(* CoDeSys 2.3 export: V4500306_ORIGINAL.EXP *)
(* Libraries: ConnectionDiagnose.lib 3.7.07 16:35:00, PLC_EposCmd.lib 23.7.04 12:26:00, STANDARD.LIB 5.6.98 12:03:02, TcBase.lib 14.5.09 12:14:08, TcBaseMath.lib 27.7.04 12:07:56, TcIoFunctions.lib 27.1.17 17:22:22, TcMath.lib 23.9.04 15:15:30, TcMC.lib 27.7.15 08:51:38, TcNC.lib 10.10.08 17:55:34, TcSystem.lib 7.6.16 11:01:22, TcUtilities.lib 3.2.16 16:08:58 *)

(* Task configuration *)
TASK Standard (PRIORITY := 0, INTERVAL := T#5ms);
PRG_STARTUP();
PRG_VISU();
PRG_PROCESS();
PRG_STATION();
PRG_HW_GENERAL();
PRG_HW_STATION();
PRG_TWINSAFE();
END_TASK
TASK Ctrl_Panel (PRIORITY := 1, INTERVAL := T#100ms);
PRG_USB_IO_PANEL();
END_TASK

(* Global variable list: Constant_Variablen *)
VAR_GLOBAL CONSTANT
	(* developpement *)
	(*sRootPLC:STRING(255):='C:';*)
	(* machine *)
	cssRootPLC:STRING(255):='';
	(* HDD *)
	csiMaxFileLine:INT:=255;
	(* Axis *)
	csiMaxAxisFileObj:INT:=50;
	ciMaxWireStretch:INT:=32767;
	(* Visualisation *)
	csiMaxPage:INT:=50;
	csiMaxUserLevel:INT:=3;
	(* Profile *)
	csiMaxProfile:INT:=100;
END_VAR

(* Global variable list: Globale_Variablen *)
VAR_GLOBAL
(* Structure layer 2 *)
	T_HDD:ST_HDD;
	T_NovRam : ST_NOVRAM;
	T_CtrlePanel:ST_CTRLEPANEL;
	T_DeviceID:ST_DEVICEID;
	T_BoxID:ST_BOXID;
	 T_AxisNodeState AT %I* :ST_NODESTATE;
(* Visualization *)
	QVisCtrl :ST_QVISCTRLE;(*~	(QVis) (InOut:2)	~*)
	T_ExchgParam :ST_QVIS_EXCHG_PARAM;(*~	(QVis) (InOut:2)	~*)
	T_VisuQVis:ST_QVIS;
(* Control Button Start/Stop *)
	T_CtrleBtStartStop:ST_CTRLEBUTTON;
(* StartUp *)
	T_StartUp:ST_STARTUP;
(* Station *)
	T_Station:ST_STATION;
(* Process *)
	T_Process : ST_PROCESS;
(* Profile *)
	T_Profile:ST_PROFILE;
(* Static Error List *)
	T_ErrorList:ST_ERROR_LIST;	(* Static define Error List *)
(* IO's *)
	IarxDigitalInput AT %I* : ARRAY[1..64] OF BOOL;
	QarxDigitalOutput AT %Q* : ARRAY[1..64] OF BOOL;
	IariAnalogInput AT %I* : ARRAY[1..32] OF INT;
	QariAnalogOutput AT %Q* : ARRAY[1..32] OF INT;
	QarxCylinder AT %Q* : ARRAY[1..32] OF BOOL;
(* TwinSafe *)
	T_TwinSafeCtrleIN AT %I*:ST_TWINSAFE_CTRLE_IN;
	T_TwinSafeCtrleOUT AT %Q*:ST_TWINSAFE_CTRLE_OUT;
	T_TwinSafeIn:ST_TWINSAFE_IN;
	T_TwinSafeOut AT %I*:ST_TWINSAFE_OUT;
END_VAR

(* Global variable list: TwinCAT_Configuration *)
(* Generated automatically by TwinCAT - (read only) *)
VAR_CONFIG
	PRG_HW_STATION.TToolLeftRxPdoPara AT %QB0 : ST_RX_PDO_PARA;
	PRG_HW_STATION.TToolLeftTxPdoPara AT %IB0 : ST_TX_PDO_PARA;
	PRG_HW_STATION.TToolCenterRxPdoPara AT %QB27 : ST_RX_PDO_PARA;
	PRG_HW_STATION.TToolCenterTxPdoPara AT %IB17 : ST_TX_PDO_PARA;
	PRG_HW_STATION.TToolRightRxPdoPara AT %QB54 : ST_RX_PDO_PARA;
	PRG_HW_STATION.TToolRightTxPdoPara AT %IB34 : ST_TX_PDO_PARA;
	PRG_HW_STATION.TToolFeederRxPdoPara AT %QB81 : ST_RX_PDO_PARA;
	PRG_HW_STATION.TToolFeederTxPdoPara AT %IB51 : ST_TX_PDO_PARA;
	PRG_HW_STATION.TGrindFeederRxPdoPara AT %QB108 : ST_RX_PDO_PARA;
	PRG_HW_STATION.TGrindFeederTxPdoPara AT %IB68 : ST_TX_PDO_PARA;
	PRG_HW_STATION.stToolLeftRefOut AT %QB135 : PLCTONC_AXLESTRUCT;
	PRG_HW_STATION.stToolLeftRefIn AT %IB85 : NCTOPLC_AXLESTRUCT;
	PRG_HW_STATION.stToolCenterRefOut AT %QB263 : PLCTONC_AXLESTRUCT;
	PRG_HW_STATION.stToolCenterRefIn AT %IB213 : NCTOPLC_AXLESTRUCT;
	PRG_HW_STATION.stToolRightRefOut AT %QB391 : PLCTONC_AXLESTRUCT;
	PRG_HW_STATION.stToolRightRefIn AT %IB341 : NCTOPLC_AXLESTRUCT;
	PRG_HW_STATION.stToolFeederRefOut AT %QB519 : PLCTONC_AXLESTRUCT;
	PRG_HW_STATION.stToolFeederRefIn AT %IB469 : NCTOPLC_AXLESTRUCT;
	PRG_HW_STATION.stGrindFeederRefOut AT %QB647 : PLCTONC_AXLESTRUCT;
	PRG_HW_STATION.stGrindFeederRefIn AT %IB597 : NCTOPLC_AXLESTRUCT;
	PRG_HW_STATION.auiActualAxisTorqueBeckhoff AT %IB725 : ARRAY [1..5] OF UINT;
	PRG_HW_STATION.axInputAxisBeckhoff AT %IB735 : ARRAY [1..5, 1..8] OF BOOL;
	PRG_TWINSAFE.TwinSAFEinputKlemme1.KLx904_SafetyIn AT %IB920 : TwinSAFE_SafetyIn;	(*  ~ {LinkedWith:TIID^CX1000_PLC^CX1100-KB^Klemme 9 (KL1904)^Kanal 1^Safety In} *)
	PRG_TWINSAFE.TwinSAFEinputKlemme2.KLx904_SafetyIn AT %IB926 : TwinSAFE_SafetyIn;	(*  ~ {LinkedWith:TIID^CX1000_PLC^CX1100-KB^Klemme 10 (KL1904)^Kanal 1^Safety In} *)
	PRG_TWINSAFE.TwinSAFEinputKlemme3.KLx904_SafetyIn AT %IB932 : TwinSAFE_SafetyIn;	(*  ~ {LinkedWith:TIID^CX1000_PLC^CX1100-KB^Klemme 11 (KL1904)^Kanal 1^Safety In} *)
	PRG_USB_IO_PANEL.IarxCtrlePanelButton AT %IB775 : ARRAY [1..10] OF BOOL;
	PRG_USB_IO_PANEL.QarxCtrlePanelLed AT %QB775 : ARRAY [1..10] OF BOOL;
	.T_AxisNodeState AT %IB940 : ST_NODESTATE;
	.IarxDigitalInput AT %IB785 : ARRAY [1..64] OF BOOL;
	.QarxDigitalOutput AT %QB785 : ARRAY [1..64] OF BOOL;
	.IariAnalogInput AT %IB849 : ARRAY [1..32] OF INT;
	.QariAnalogOutput AT %QB849 : ARRAY [1..32] OF INT;
	.QarxCylinder AT %QB913 : ARRAY [1..32] OF BOOL;
	.T_TwinSafeCtrleIN AT %IB913 : ST_TWINSAFE_CTRLE_IN;
	.T_TwinSafeCtrleOUT AT %QB945 : ST_TWINSAFE_CTRLE_OUT;
	.T_TwinSafeOut AT %IB916 : ST_TWINSAFE_OUT;
END_VAR

(* Data type in AXIS *)
TYPE ST_AXIS :
STRUCT
	T_CtrleSingle:ST_CTRLESINGLE;
	T_CtrleMulti:ST_CTRLEMULTI;
	T_ParamFileObj:ARRAY[1..40] OF ST_PARAM_FILE_OBJ;
	T_Config_Gen:ST_CONFIG_GENERAL;
	T_Config_ObjFileValue:ST_CONFIG_OBJECT;	(* Gilt nicht für Ecostep *)
 	T_Config_Setting:ST_CONFIG_SETTING;			(* Gilt nicht für Ecostep *)
	T_LiveValue:ST_LIVEVALUE;
	T_Oscillation:ST_OSCILLATION;					(* Gilt nicht für Ecostep *)
	T_Torque:ST_AXISTORQUE;					(* Gilt nicht für Ecostep *)
	T_FileObj:ST_AXIS_FILE_OBJ;
	T_RxPdoParameter:ST_RX_PDO_PARA;
	T_TxPdoParameter:ST_TX_PDO_PARA;
	T_SoftwareDetails:ST_SOFTWARE_INFO;
END_STRUCT
END_TYPE

(* Data type in AXIS *)
TYPE ST_AXIS_FILE_OBJ :
STRUCT
	sData: ARRAY[1..csiMaxAxisFileObj] OF STRING(120);
END_STRUCT
END_TYPE

(* Data type in AXIS *)
TYPE ST_AXISTORQUE :
STRUCT
(* input *)
	xActive:BOOL;
(* output *)
	rAverage:REAL;
	rMinAverage:REAL;
	rMaxAverage:REAL;
	rLastValue:REAL;
	rMinValue:REAL;
	rMaxValue:REAL;
	iSensitivity:INT;
	rMaxVariationSpindle:REAL;
	rActualVariationSpindle:REAL;
END_STRUCT
END_TYPE

(* Data type in AXIS *)
TYPE ST_CONFIG_GENERAL :
STRUCT
	sDeviceName:STRING(32);
	sDeviceFileName:STRING(32);
	sFileNamePDOMapping:STRING(32);
	sServoNetId:STRING(23);		(* Beckhoff *)
	sAmsNetId:T_AmsNetId;		(* Ecostep *)
	udiNC_TaskIdxGrp:UDINT;		(* Beckhoff *)
	udiNodeId:UDINT;				(* Ecostep *)
	iTyp:INT;
	iMachineType:INT;			(* 1 = MicroWire, 2 = MicroRod *)
END_STRUCT
END_TYPE

(* Data type in AXIS *)
TYPE ST_CONFIG_OBJECT :
STRUCT
(* Object value *)
	lrMaxVelocity:LREAL;
	lrCalVelocityForward:LREAL;
	lrCalVelocityBackward:LREAL;
	lrAcceleration:LREAL;
	lrDecceleration:LREAL;
	lrJerk:LREAL;
	xSWLimitPos:BOOL;
	xHWLimitPos:BOOL;
	lrSWLimitPos:LREAL;
	xSWLimitNeg:BOOL;
	xHWLimitNeg:BOOL;
	lrSWLimitNeg:LREAL;
	lrScaleFactor:LREAL;
END_STRUCT
END_TYPE

(* Data type in AXIS *)
TYPE ST_CONFIG_SETTING :
STRUCT
	lrJogFast:LREAL;
	lrJogSlow:LREAL;
	lrJogStepFast:LREAL;
	lrJogStepSlow:LREAL;
	lrVelocityAbs:LREAL;
	lrVelocityRel:LREAL;
	lrVelocityProcess:LREAL;
	lrSpindleCurrentLimit:LREAL;
	xHardwareLimitPos:BOOL;
	xHardwareLimitNeg:BOOL;
	lrHWLimitDecceleration:LREAL;
	rHCRampDeceleration:REAL;
	rHCRampJerk:REAL;
END_STRUCT
END_TYPE

(* Data type in AXIS *)
TYPE ST_CTRLEMULTI :
STRUCT
(* Input *)
	xExecute:BOOL:=FALSE;
	xReset:BOOL:=FALSE;
	iNumerator:INT:=1;
	uiDenominator:UINT:=1;
	iFunction:INT:=0;

(* Ouput *)
	xDone:BOOL:=FALSE;
	xErr:BOOL:=FALSE;
	udiErrorID:UDINT:=0;
END_STRUCT
END_TYPE

(* Data type in AXIS *)
TYPE ST_CTRLESINGLE :
STRUCT
(* Input *)
	xExecute:BOOL:=FALSE;
	iFunction:INT:=0;
	xReset:BOOL:=FALSE;
	iInput:INT:=0;
	lrPosition:LREAL:=0;
	lrDistance:LREAL:=0;
	lrVelocity:LREAL:=0;
	lrAcceleration:LREAL:=0;
	lrDecceleration:LREAL:=0;
	lrJerk:REAL:=0;
	dwOverride:DWORD:=100;
	rSetPosition:REAL:=0;
	rSetTorque:REAL:=0;
	sSend:STRING(20):='';
	lrScaleFactor:LREAL:=0;
	lrGearRatioFactor:LREAL:=0;
	lrGearRatioDivider:LREAL:=0;
	lrGearRatio:LREAL:=0;	(* calculate lrGearRatioFactor / lrGearRatioDivider *)
	iModuloDirection:INT;		(*	Enum Werte:
									 MC_Positive_Direction := 1,
    									MC_Shortest_Way :=2,
    									MC_Negative_Direction :=3,
    									MC_Current_Direction :=4
							*)
	lrHomingMethode:LREAL;
	lrHomeOffset:LREAL;
	lrHomeSpeedSwitch:LREAL;
	lrHomeSpeedZero:LREAL;
	lrHomeAcceleration:LREAL;
	lrGearFactor:LREAL;
	lrGearDivider:LREAL;
	lrSWNegLimitSwitch:LREAL;
	lrSWPosLimitSwitch:LREAL;
	xBlockAcclDeclParameter:BOOL;

(* Output *)
	xDone:BOOL:=FALSE;
	xErr:BOOL:=FALSE;
	udiErrorID:UDINT:=0;
	xPower:BOOL:=FALSE;
	xReady:BOOL:=FALSE;
	xNotMoving:BOOL:=FALSE;
	xRef:BOOL:=FALSE;
	xSlave:BOOL:=FALSE;
	xConstantVel:BOOL:=FALSE;
	xBusyNewPosAndVel:BOOL:=FALSE;
	xDriveTorque:BOOL:=FALSE;
	iOutput:INT:=0;
	xSWLimitPos:BOOL:=FALSE;
	xSWLimitNeg:BOOL:=FALSE;
	xHWLimitPos:BOOL:=FALSE;
	xHWLimitNeg:BOOL:=FALSE;
	xSpindleBlocked:BOOL:=FALSE;
	iStrokeAngleRefIndex:INT;	(* Gilt für die Prozedur für das einstellen des Referenzindex der Achse *)
END_STRUCT
END_TYPE

(* Data type in AXIS *)
TYPE ST_LIVEVALUE :
STRUCT
	dwState:DWORD;
	uiActualTorque:UINT;
	diActualTorqueCalc:DINT;	(* entsricht dem uiActualTorque, nur dass positiver und negativer Torque berücksichtigt wird *)
	lrActualVelocity:LREAL;
	lrActualPosition:LREAL;
	bDigitalInput:BYTE;
	lrSollPosition:LREAL;
	lrActualPositionNotModulo:LREAL;
	lrActualPositionRelativ:LREAL;
END_STRUCT
END_TYPE

(* Data type in AXIS *)
TYPE ST_NODESTATE :
STRUCT
	bToolLeftNodeState:BYTE;
	bToolCenterNodeState:BYTE;
	bToolRightNodeState:BYTE;
	bToolFeederNodeState:BYTE;
	bGrindFeederNodeState:BYTE;
END_STRUCT
END_TYPE

(* Data type in AXIS *)
TYPE ST_OSCILLATION :
STRUCT
	rFrequence:REAL;
	rOffset:REAL;
	rPosTorqueLimitOffset:REAL;
	iCycle:INT;
END_STRUCT
END_TYPE

(* Data type in AXIS *)
TYPE ST_PARAM_FILE_OBJ :
STRUCT
	udiIdxGroup:UDINT:=0;
	udiIndexOffset:UDINT:=0;
	udiLength:UDINT:=0;
	lrReal:LREAL:=0;
	sName:STRING(20);
END_STRUCT
END_TYPE

(* Data type in AXIS *)
TYPE ST_RX_PDO_PARA :
STRUCT
	udiProfileVelocity:UDINT;
	diTargetVelocity:DINT;
	udiProfileDeceleration:UDINT;
	udiProfileAcceleration:UDINT;
	diTargetPosition:DINT;
	iGearFactor:INT;
	uiGearDivider:UINT;
	iControlWord:INT;
	siOperationModes:SINT;
END_STRUCT
END_TYPE

(* Data type in AXIS *)
TYPE ST_SOFTWARE_INFO :
STRUCT
	lrSoftwareVersion:REAL;
	lrBuildVersion:REAL;
	lrDateCode:REAL;
	sDateCode:STRING;
END_STRUCT
END_TYPE

(* Data type in AXIS *)
TYPE ST_TX_PDO_PARA :
STRUCT
	diActualPosition:DINT;
	diActualVelocity:DINT;
	uiStatusWord:UINT;
	iActualCurrent:INT;
	udiDigitalInput:UDINT;
	siOperationModesDisplay:SINT;
END_STRUCT
END_TYPE

(* Data type in CX1020 *)
TYPE ST_BOXID :
STRUCT
(* control structure *)
	T_Ctrle:ST_CTRLE_DEVICEID;
(* Data *)
	(* servo Beckhoff-->Lightbus *)
	T_Servo_ToolLeft:ST_BOXID_DATA_ADR;
	T_Servo_ToolCenter:ST_BOXID_DATA_ADR;
	T_Servo_ToolRight:ST_BOXID_DATA_ADR;
	T_Servo_ToolFeeder:ST_BOXID_DATA_ADR;
	T_Servo_GrindFeeder:ST_BOXID_DATA_ADR;
END_STRUCT
END_TYPE

(* Data type in CX1020 *)
TYPE ST_BOXID_DATA_ADR :
STRUCT
	sDeviceName:T_MaxString;
	sBoxName:T_MaxString;
	xDeviceOption:BOOL;
	wAddrBox:WORD;
	sAmsNetId:T_AmsNetId;
END_STRUCT
END_TYPE

(* Data type in CX1020 *)
TYPE ST_CTRLE_DEVICEID :
STRUCT
(* input *)
	xExecute:BOOL:=FALSE;
	xReset:BOOL:=FALSE;
	xLocked:BOOL:=FALSE;
(*
	iStationNr:INT:=0;
	iStationType:INT:=0;
	iSpindleType:INT:=0;
*)
	iMachineType:INT:=0;

(* output *)
	xDone:BOOL:=FALSE;
	xErr:BOOL:=FALSE;
	udiErrorID:UDINT:=0;

END_STRUCT
END_TYPE

(* Data type in CX1020 *)
TYPE ST_DEVICEID :
STRUCT
(* control structure *)
	T_Ctrle:ST_CTRLE_DEVICEID;
(* Data *)
	(* PLC *)
		T_CX1020:ST_DEVICEID_DATA_ADR;
	(* feldbus *)
		T_CANOpenMaster:ST_DEVICEID_DATA_ADR;
		T_LightbusMaster:ST_DEVICEID_DATA_ADR;
	(* NovRAM *)
		T_NovRAM:ST_DEVICEID_DATA_ADR;
END_STRUCT
END_TYPE

(* Data type in CX1020 *)
TYPE ST_DEVICEID_DATA_ADR :
STRUCT
	sDeviceName:T_MaxString;
	xDeviceOption:BOOL;
	udiDeviceID:UDINT;
	sAmsNetId:T_AmsNetId;
END_STRUCT
END_TYPE

(* Data type in Cylinder *)
TYPE ST_ANALOG :
STRUCT
(* input *)
	tDelayActiv:TIME;
	iAnalogIN:INT;
	rForceIn:REAL;
	iRampFctOn:INT;
	iRampFctOff:INT;
	rStepValue:REAL;
	rLengthIn:REAL;
(* Output *)
	xActiv:BOOL;
	iAnalogOut:INT;
	rForceOut:REAL;
	tTimeActivOn:TIME;
	tTimeActivOff:TIME;
END_STRUCT
END_TYPE

(* Data type in Cylinder *)
TYPE ST_ANALOG_CYL :
STRUCT
(* input *)
	tDelayActiv:TIME;
	iAnalogIN:INT;
	rForceIn:REAL;
(* Output *)
	xActiv:BOOL;
	iAnalogOut:INT;
	rForceOut:REAL;
END_STRUCT
END_TYPE

(* Data type in Cylinder *)
TYPE ST_CONFIG :
STRUCT
	tDelayOn:TIME;
	tDelayOff:TIME;
	tDelayPreOn:TIME;
	tDelayPreOff:TIME;
	xCtrlePosOn:BOOL;
	xCtrlePosOff:BOOL;
	tTimeOut:TIME;
	xActivState:BOOL;
END_STRUCT
END_TYPE

(* Data type in Cylinder *)
TYPE ST_CTRLECYL :
STRUCT
(* input *)
	xFBActiv:BOOL;
	xExecute:BOOL;
	xReset:BOOL;
	iFunction:INT;
(* output *)
	xDone:BOOL;
	xErr:BOOL;
	udiErrorID:UDINT;
	xStatePosOn:BOOL;
	xStatePosOff:BOOL;
	T_AnalogCylinder:ST_ANALOG_CYL;
	T_Standard:ST_STANDARD;
	T_Analog:ST_ANALOG;
END_STRUCT
END_TYPE

(* Data type in Cylinder *)
TYPE ST_CYLINDER :
STRUCT
	T_Config:ST_CONFIG;
	T_CtrleCyl:ST_CTRLECYL;
END_STRUCT
END_TYPE

(* Data type in Cylinder *)
TYPE ST_STANDARD :
STRUCT
(* Input *)
	tDelayActiv:TIME;
	tDelayAfterSensor:TIME;
(* Output *)
	xActivOn:BOOL;
	xActivOff:BOOL;
END_STRUCT
END_TYPE

(* Data type in Geometry *)
TYPE ST_GEOMETRY :
STRUCT
	arStartDiameter: ARRAY [1..6] OF REAL;
	arEndDiameter: ARRAY [1..6] OF REAL;
	arSectionLength: ARRAY [1..6] OF REAL;
	arSectionPitch: ARRAY [1..6] OF REAL;
	axActiveSection:ARRAY [1..6] OF BOOL;
END_STRUCT
END_TYPE

(* Data type in Geometry *)
TYPE ST_GEOMETRY_COMMON :
STRUCT
	abSectionSelectForm:ARRAY [1..6] OF BYTE; (* 0=Disactivate Section, 1=Zylindre large, 2=Zylindre small, 3=Cone Negative, 4=Cone Positive *)
	wWrongInput:WORD;
	wWrongInput_2:WORD;
	rMinToolDiameter:REAL;
	rMaxToolDiameter:REAL;
	rMinToolLength:REAL;
	rMaxToolLength:REAL;
	T_Geometry:ST_GEOMETRY;
END_STRUCT
END_TYPE

(* Data type in HDD *)
TYPE ST_CTRLE_HDD :
STRUCT
(* input *)
	xExecute:BOOL:=FALSE;
	xReset:BOOL:=FALSE;
	iFunction:INT:=0;
	tTimeOut:TIME;
	xLocked:BOOL:=FALSE;

(* output *)
	xDone:BOOL:=FALSE;
	xErr:BOOL:=FALSE;
	udiErrorID:UDINT:=0;
END_STRUCT
END_TYPE

(* Data type in HDD *)
TYPE ST_HDD :
STRUCT
	T_Ctrle:ST_CTRLE_HDD;
	T_Config:ST_HDD_CONFIG;
	T_File:ST_HDD_FILE;
	T_Data:ST_HDD_DATA;
END_STRUCT
END_TYPE

(* Data type in HDD *)
TYPE ST_HDD_CONFIG :
STRUCT
	sNetId:T_AmsNetId;
END_STRUCT
END_TYPE

(* Data type in HDD *)
TYPE ST_HDD_DATA :
STRUCT
	sData: ARRAY[1..csiMaxFileLine] OF STRING(255);
END_STRUCT
END_TYPE

(* Data type in HDD *)
TYPE ST_HDD_FILE :
STRUCT
	sPathAndFileName:STRING(255):='';
	sOldPathAndFileName:STRING(255):='';
	dwPtrWriteBuffer:DWORD:=0;
	udiLenBuffer:UDINT:=0;
END_STRUCT
END_TYPE

(* Data type in Panel *)
TYPE ST_CTRLEPANEL :
STRUCT
(* Input *)
	xExecute:BOOL:=FALSE;
	iFunction:INT:=0;
	xReset:BOOL:=FALSE;
(* output *)
	xDone:BOOL;
	xErr:BOOL;
	udiErrorID:UDINT;
	udiButton:UDINT:=0;
	udiLED:UDINT:=0;
END_STRUCT
END_TYPE

(* Data type in Process *)
TYPE ST_FCTPROCESS :
STRUCT
	xEnable : BOOL :=FALSE;
	xStart: BOOL := FALSE;
	xStop: BOOL := FALSE;
	xStopCycle : BOOL :=FALSE;
	xQuitErr : BOOL := FALSE;
	xAbord : BOOL := FALSE;
	xProcessHold : BOOL;
	xEnd : BOOL := FALSE;
	xError : BOOL := FALSE;
	diErrorNr : DINT := 0;
END_STRUCT
END_TYPE

(* Data type in Process *)
TYPE ST_PARA_WARMUP :
STRUCT
	iWarmUp_TimeON_Hour		:INT;
	iWarmUp_TimeON_Minute		:INT;
	iWarmUp_TimeOFF_Hour		:INT;
	iWarmUp_TimeOFF_Minute		:INT;
	axDayOfWeek				:ARRAY [0..7] OF BOOL;	(* 0=Sonntag, 1=Montag..usw *)

(*SOA 30.01.23 *)
	iWarmUp_TimeDIF_Hour		:INT;
	iWarmUp_TimeDIF_Minute		:INT;
END_STRUCT
END_TYPE

(* Data type in Process *)
TYPE ST_PROCESS :
STRUCT
	iFunctNr : INT :=0;
	xEnable : BOOL := FALSE;
	xStart : BOOL := FALSE;
	xEnd : BOOL := FALSE;
	xStop : BOOL := FALSE;
	xStopCycle : BOOL :=FALSE;
	xRdy : BOOL := FALSE;
	xError : BOOL := FALSE;
	diErrorNr : DINT :=0;
	xQuitError : BOOL := FALSE;
	xProcessHold : BOOL;
	wStatus : WORD := 0;
	xAbord : BOOL := FALSE;
	xReferenced : BOOL := FALSE;
	TFctProcess : ST_FCTPROCESS;
END_STRUCT
END_TYPE

(* Data type in Profile *)
TYPE ST_PROFILE :
STRUCT
	T_Ctrle:ST_PROFILE_CTRLE;
	T_Id:ST_PROFILE_ID;
	(*T_DataOnline:ST_PROFILEONLINECHANGE;*)
END_STRUCT
END_TYPE

(* Data type in Profile *)
TYPE ST_PROFILE_CTRLE :
STRUCT
(* input *)
	xExecute:BOOL:=FALSE;
	xReset:BOOL:=FALSE;
	iFunction:INT:=0;

(* Output *)
	xDone:BOOL:=FALSE;
	xErr:BOOL:=FALSE;
	udiErrorID:UDINT:=0;
END_STRUCT
END_TYPE

(* Data type in Profile *)
TYPE ST_PROFILE_ID :
STRUCT
	iNumber:INT;
	sName:STRING(30);
END_STRUCT
END_TYPE

(* Data type in Profile *)
TYPE ST_PROFILE_LIST :
STRUCT
	iNumber:INT;
	sName:STRING(30);
END_STRUCT
END_TYPE

(* Data type in Profile *)
TYPE ST_PROFILE_LIST_MANAGE :
STRUCT
	xListProfileUp:BOOL;
	xListProfileDown:BOOL;
	xListProfileUpFast:BOOL;
	xListProfileDownFast:BOOL;
END_STRUCT
END_TYPE

(* Data type in QVis *)
TYPE ST_BUTTON :
STRUCT
	xInputState:BOOL;
	xLedState:BOOL;
	xResetTime:BOOL;
	tPressTime:TIME;
END_STRUCT
END_TYPE

(* Data type in QVis *)
TYPE ST_CONFIGPAGE :
STRUCT
	sName:STRING(32);
	wMaskBtPanelLeft:WORD;
	wMaskBtPanelRight:WORD;
	wMaskFunctionPanel:WORD;
	wMaskTouchScreenNavPanel:WORD;
	(* active movement mask *)
	wMaskActiveMachineBtPanelLeft:WORD;
	wMaskActiveMachineBtPanelRight:WORD;
	wMaskActiveMachineFunctionPanel:WORD;
	wMaskActiveMachineNavPanel:WORD;
	(* functions *)
	aiRTrigActionPanelRight:ARRAY[1..5] OF INT:=5(0);
	aiFTrigActionPanelRight:ARRAY[1..5] OF INT:=5(0);
	aiDelayActionPanelRight:ARRAY[1..5] OF INT:=5(0);
	aiRTrigActionFunctionPanel:ARRAY[1..12] OF INT:=12(0);
	aiFTrigActionTouchScreenNavPanel:ARRAY[1..6] OF INT:=6(0);
	(* start/stop button *)
	xMaskBtStart:BOOL;
	xMaskBtStop:BOOL;
END_STRUCT
END_TYPE

(* Data type in QVis *)
TYPE ST_CTRLEACTION :
STRUCT
(* Input *)
	xExecute:BOOL;
	xReset:BOOL;
	iFunction:INT;
	xResetParaListValue:BOOL;
(* Output *)
	xDone:BOOL;
	xNotReady:BOOL;
	xErr:BOOL;
	udiErrorID:UDINT;
END_STRUCT
END_TYPE

(* Data type in QVis *)
TYPE ST_CTRLEBUTTON :
STRUCT
	T_Start:ST_BUTTON;
	T_Stop:ST_BUTTON;
END_STRUCT
END_TYPE

(* Data type in QVis *)
TYPE ST_CTRLEPROCESS :
STRUCT
(* Input *)
	xExecute:BOOL;
	xReset:BOOL;
	iFunction:INT;
(* Output *)
	xDone:BOOL;
	xErr:BOOL;
	udiErrorID:UDINT;
END_STRUCT
END_TYPE

(* Data type in QVis *)
TYPE ST_CTRLEVISU :
STRUCT
(* Input *)
	xActive:BOOL;
	xExecute:BOOL;
	xReset:BOOL;
	iFunction:INT;
(* Output *)
	xDone:BOOL;
	xErr:BOOL;
	udiErrorID:UDINT;
	xQvis:BOOL;
END_STRUCT
END_TYPE

(* Data type in QVis *)
TYPE ST_EXCHG_BTFUNCTIONPANEL :
STRUCT
	wState:WORD;
	wActivBt:WORD;
	wNotMasktext:WORD;
	bF1SelectText:BYTE;
	bF2SelectText:BYTE;
	bF3SelectText:BYTE;
	bF4SelectText:BYTE;
	bF5SelectText:BYTE;
	bF6SelectText:BYTE;
	bF7SelectText:BYTE;
	bF8SelectText:BYTE;
	bF9SelectText:BYTE;
	bF10SelectText:BYTE;
	bF11SelectText:BYTE;
	bF12SelectText:BYTE;
END_STRUCT
END_TYPE

(* Data type in QVis *)
TYPE ST_EXCHG_CONFIG :
STRUCT
	xNoTouchScreenBtPanel:BOOL;
	iEditParam:INT;
	xBlockParaListNavi:BOOL;
	xBlockParaListNavi1:BOOL;
	xBlockNavParaList:BOOL;
	xBlockNavParaListTeachRot:BOOL;
	xBlockProfilList:BOOL;
	iSelectParaList:INT;
	iSelectParaListTeachRot:INT;
END_STRUCT
END_TYPE

(* Data type in QVis *)
TYPE ST_EXCHG_CYLINDER :
STRUCT
(*	iSelectCylToolTension:INT; *)
	xToolTension:BOOL;
	bPosToolTension:BYTE;

	T_ParamToolTension:ST_EXCHG_PARAM_CYL_FORCE;
	iSelectToolTensionForce:INT;
	rToSetToolTensionForce:REAL;
(*22.12.2009: KFS	{	*)
	iSelectCylinder_Sonder1:INT;

	xCylToolLeft:BOOL;
	bPosCylToolLeft:BYTE;

	xCylToolRight:BOOL;
	bPosCylToolRight:BYTE;

	xCylToolCenter:BOOL;
	bPosCylToolCenter:BYTE;

	xCylToolPrismaLeft:BOOL;
	bPosCylToolPrismaLeft:BYTE;

	xCylToolPrismaRight:BOOL;
	bPosCylToolPrismalRight:BYTE;
(*22.12.2009: KFS	}	*)
END_STRUCT
END_TYPE

(* Data type in QVis *)
TYPE ST_EXCHG_FUNCTION_COMMON :
STRUCT
	(* Overlay for input measured Tool diameter *)
	xOpenOverlayMeasureInput:BOOL;
	(* Overlay for input the correction of the GrindFeeder Plunge *)
	xOpenOverlaySetGrindPlunge:BOOL;
	(* Overlay for open a Messagebox *)
	xOpenOverlayMessageBox:BOOL;
	sMessageBoxLine1:STRING(50);
	sMessageBoxLine2:STRING(50);
	sMessageBoxLine3:STRING(50);
	sMessageBoxLine4:STRING(50);
	sMessageBoxLine5:STRING(50);
	sMessageBoxLine6:STRING(50);
	xSaveButton:BOOL;
	xExitButton:BOOL;
	rInputMeasToolDiameter:REAL;
	rInputGrindPlunge:REAL;
	xHideProgressbar:BOOL;

	(*SOA 12.01.2023 { *)
	(* Setup WarmUp *)
	TWarmUp_Para						:ST_PARA_WARMUP;
	axWarmUp_DayOfWeekButton			:ARRAY [0..6] OF BOOL;	(* 0=Sonntag, 1=Montag..usw *)
	xWarmUp_ContactorMachine_Active		:BOOL;
	xWarmUp_MessageWarning			:BOOL;	(* Mittels dieser Meldung wird hingewiesen dass die Maschine nächstens eingeschaltet wird *)
	xWarmUp_MessageWarning_2			:BOOL;	(* Mittels dieser Meldung wird gefragt, ob die Maschine wirklich eingeschaltet werden soll *)
	iWarmUp_ColourChange				:BOOL;
	(*SOA 12.01.2023 } *)

END_STRUCT
END_TYPE

(* Data type in QVis *)
TYPE ST_EXCHG_INFO_PROCESS :
STRUCT
	iProfile:INT;
	sProfileName:STRING(30);
	xOnlineValueModified:BOOL;
END_STRUCT
END_TYPE

(* Data type in QVis *)
TYPE ST_EXCHG_INFOVALUE_COMMON :
STRUCT
	rActualGrindAxisPosition:REAL;
	rActualGrindAxisSpeed:REAL;
	rActualToolRotSpeed:REAL;
	rActualWireFeedPosition:REAL;
	rActualWireFeedSpeed:REAL;
	rActualToolLeftTorque:REAL;
	rCalculToolLeftTorque:REAL;
	rActualToolCenterTorque:REAL;
	rCalculToolCenterTorque:REAL;
	rActualToolRightTorque:REAL;
	rCalculToolRightTorque:REAL;
	rToolLengthCalibration:REAL;
	rToolDiameter:REAL;
	rToolTotalLength:REAL;
	rPitchCalibration:REAL;
	rToolTensionForce:REAL;
	iTotalCountDownCycle:INT;
	iCountDownCycle:INT;
	iTotalCountDownPlungeCycle:INT;
	iCountDownPlungeCycle:INT;
	iTotalCountDownGrooveCycle:INT;
	iCountDownGrooveCycle:INT;
	tAutoTimeTotal:TIME;
	tAutoTimeLeft:TIME;

	rCorrectionToolDiameter:REAL;
	xKeyPadActivation:BOOL;

	(* Progressbar for Tool Calibration *)
	bProgressbarToolCalibration:BYTE;
	bProgressbarAutoGeometry:BYTE;
	bProgressbarAutoGroove:BYTE;

	(* Effectiv working geometry *)
	arStartDiameter: ARRAY [1..6] OF REAL;
	arEndDiameter: ARRAY [1..6] OF REAL;
	(* Part State display *)
	bActivePartNumber:BYTE;

END_STRUCT
END_TYPE

(* Data type in QVis *)
TYPE ST_EXCHG_LEVEL :
STRUCT
	iActLevel:INT;
	iPwSystem:INT;
	iRandom:INT;
END_STRUCT
END_TYPE

(* Data type in QVis *)
TYPE ST_EXCHG_MACHINE :
STRUCT
	iFunction:INT;
	udiState_Input:UDINT;
	T_Process:ST_EXCHG_PROCESS;
END_STRUCT
END_TYPE

(* Data type in QVis *)
TYPE ST_EXCHG_MESSAGE :
STRUCT
	iState:INT;
	iStateBIOS:INT;
	sDynamicTextEnglish:STRING(100);
	sDynamicTextDeutsch:STRING(100);
	sDynamicTextFrancais:STRING(100);
END_STRUCT
END_TYPE

(* Data type in QVis *)
TYPE ST_EXCHG_MESSAGE_ERROR :
STRUCT
	asMsgErrorList:ARRAY [1..20] OF STRING(100);
END_STRUCT
END_TYPE

(* Data type in QVis *)
TYPE ST_EXCHG_PARAM_AUTOGEOMETRY :
STRUCT
	rPlungeLengthToolFeedGeometry:REAL;
	rPlungeSpeedGrindFeedGeometry:REAL;
	rDisplaceLengthToolFeedGeometry:REAL;
	rDisplaceSpeedGrindFeedGeometry:REAL;
	xPlungeActivationGeometry:BOOL;
	xDisplaceActivationGeometry:BOOL;
	iCycleGeometry:INT;
	rPlungeCycleGrindFeedGeometry:REAL;
	rSpeedToolRotationGeometry:REAL;
(*08.07.2014: KFS	{	*)
	xWarmUp:BOOL;
(*08.07.2014: KFS	}	*)
	 xMoveTableStuderBW:BOOL;  (*SOA *)
END_STRUCT
END_TYPE

(* Data type in QVis *)
TYPE ST_EXCHG_PARAM_AUTOGROOVE :
STRUCT
	rPlungeLengthToolFeedGroove:REAL;
	rPlungeSpeedGrindFeedGroove:REAL;
	rDisplaceLengthToolFeedGroove:REAL;
	rDisplaceSpeedGrindFeedGroove:REAL;
	xPlungeActivationGroove:BOOL;
	xDisplaceActivationGroove:BOOL;

	rPitchGroove:REAL;
	rSpeedToolRotationGroove:REAL;
	xBlockGrindFeeder:BOOL;
	(*20091207 Number of grooves*)
	iNumberOfGrooves:INT;
END_STRUCT
END_TYPE

(* Data type in QVis *)
TYPE ST_EXCHG_PARAM_CALIBRATION :
STRUCT
	rPlungeLengthToolFeedCalib:REAL;
	rPlungeSpeedGrindFeedCalib:REAL;
	rDisplaceLengthToolFeedCalib:REAL;
	rDisplaceSpeedGrindFeedCalib:REAL;
	xPlungeActivationCalib:BOOL;
	xDisplaceActivationCalib:BOOL;

	rPitchCalib:REAL;
	rSpeedToolRotationCalib:REAL;
	rPlungeLengthGrindFeedCalib:REAL;
	rToolLengthCylinderPartCalib:REAL;
	rStartPosToolFeedCalib:REAL;
	rMeasurePosToolFeedCalib:REAL;	(* Für MicroRod *)
	rMeasureOffsetToolFeedCalib:REAL; (* Für MicroWire *)
END_STRUCT
END_TYPE

(* Data type in QVis *)
TYPE ST_EXCHG_PARAM_CYL_FORCE :
STRUCT
	rForce:REAL;
END_STRUCT
END_TYPE

(* Data type in QVis *)
TYPE ST_EXCHG_PARAM_MACHINE_CONFIG :
STRUCT
	iConfigMachineType:INT;
	iConfigAxisType:INT;
	iConfigVisuNavigation:INT;
	rConfigMaxToolLength:REAL;
	rConfigMaxToolLengthOriginal:REAL;
END_STRUCT
END_TYPE

(* Data type in QVis *)
TYPE ST_EXCHG_PARAM_POSITION :
STRUCT
	rLoadPosToolFeedAuto:REAL;
END_STRUCT
END_TYPE

(* Data type in QVis *)
TYPE ST_EXCHG_PARAM_PRISM :
STRUCT
	rPrismaDistanceD1:REAL;
	rPrismaDistanceD2:REAL;
	rPrismaAngleA:REAL;
	rToolDiameterMin:REAL;
	rToolDiameterMax:REAL;
	bStateInputPrisma:BYTE;	(* 0= 3 value prisma, 1 = 3 value prisma input para, 2 = 2 value prisma, 3 = 2 value prisma input para *)
	rPrismaFactor:REAL;
END_STRUCT
END_TYPE

(* Data type in QVis *)
TYPE ST_EXCHG_PARAM_PROCESS :
STRUCT
	rStartPosToolFeedAuto:REAL;
	rSpeedForwardFastGrindFeed:REAL;
	rSpeedForwardSlowGrindFeed:REAL;
	rSpeedBackwardGrindFeed:REAL;
	rToolTensionProcess:REAL;
	rToolDiameterProcess:REAL;
	rSecurityPosGrindFeedProcess:REAL;
	rOffsetBeforeToolDiaGrindFeedProcess:REAL;
	rSpeedStartPosToolFeedProcess:REAL;
	rStartPosAutoGrooveToolRotation:REAL;
END_STRUCT
END_TYPE

(* Data type in QVis *)
TYPE ST_EXCHG_PARAM_TEACHIN :
STRUCT
	rIncSlow:REAL;
	rIncFast:REAL;
	rVelSlow:REAL;
	rVelFast:REAL;
	rRefPosition:REAL;
	rRefSpeed:REAL;
	rPositionSpeed:REAL;
	rAcceleration:REAL;
	rDeceleration:REAL;
	rOffsetSWPosEndSwitch:REAL;
END_STRUCT
END_TYPE

(* Data type in QVis *)
TYPE ST_EXCHG_PARAM_TOOLTENSIONSYSTEM :
STRUCT
	rPistonDiameterTT:REAL;		(* the piston diameter of the clinder ToolTension  *)
	rPistonDiameterTT2:REAL;		(* the piston diameter of the cylinder ToolTension (Kolbenstange)*)
	rAirPressureTT:REAL;			(* max air pressure of the servo ventil *)
	rMaxForceTT:REAL;			(* calculated max. force of the ToolTension *)
	rFactorForce:REAL;			(* gear ratio of cylinder *)
END_STRUCT
END_TYPE

(* Data type in QVis *)
TYPE ST_EXCHG_PROCESS :
STRUCT
	wState:WORD;
END_STRUCT
END_TYPE

(* Data type in QVis *)
TYPE ST_EXCHG_PROFILE_COMMON :
STRUCT
(* State *)
	xImportProzessData:BOOL:=FALSE;
(* Array *)
	T_Id:ST_PROFILE_ID;
	T_ProfileManage:ST_PROFILE_LIST_MANAGE;
	T_ProfileList:ARRAY[1..10] OF ST_PROFILE_LIST;
END_STRUCT
END_TYPE

(* Data type in QVis *)
TYPE ST_EXCHG_SAFETY_CTRL :
STRUCT
	bStateMessageError:BYTE;
	bStateMessageWarning:BYTE;
	bStateMessageInfo:BYTE;
	xConfirmMsgError:BOOL;
	xConfirmMsgWarning:BOOL;
	xConfirmMsgInfo:BOOL;
	iMsgErrorLine1:INT;
	iMsgErrorLine2:INT;
	iMsgErrorLine3:INT;
	iMsgErrorLine4:INT;
	iMsgInfoLine1:INT;
	iMsgInfoLine2:INT;
	iMsgInfoLine3:INT;
	iMsgInfoLine4:INT;
	iStateStartPage:INT;
	xSetForceError:BOOL;
	diSetForceErrorNr:DINT;
	(* State Function *)
	bStateToolCalibration:BYTE;
	bStateToolTorque:BYTE;
	bStateAutoGeometry:BYTE;
	bStateAutoGroove:BYTE;
	bStateReference:BYTE;
	bStateTeachInToolLeft:BYTE;
	bStateTeachInToolCenter:BYTE;
	bStateTeachInToolRight:BYTE;
	bStateTeachInToolFeeder:BYTE;
	bStateTeachInGrindFeeder:BYTE;
	bStateReferenceMaxToolLength:BYTE;
	xBlockVisuObject:BOOL;
END_STRUCT
END_TYPE

(* Data type in QVis *)
TYPE ST_EXCHG_STATION_COMMON :
STRUCT
	(* Parameter *)
	T_InfoProcess:ST_EXCHG_INFO_PROCESS;
	T_ParamToolTensionSystem:ST_EXCHG_PARAM_TOOLTENSIONSYSTEM;
	T_PrismPara:ST_EXCHG_PARAM_PRISM;
	T_ProcessPara:ST_EXCHG_PARAM_PROCESS;
	T_AutoGeometryPara:ST_EXCHG_PARAM_AUTOGEOMETRY;
	T_AutoGroovePara:ST_EXCHG_PARAM_AUTOGROOVE;
	T_CalibrationPara:ST_EXCHG_PARAM_CALIBRATION;

	(* State Machine *)
	bStateMachine:BYTE;
	bStateMachineLED:BYTE;

	(* State Axis*)
	wState:DWORD;
	bStateAxisReelLeft:BYTE;
	bStateAxisReelCenter:BYTE;
	bStateAxisReelRight:BYTE;
	bStateAxisWireFeeder:BYTE;
	bStateAxisGrind:BYTE;

	(* State Cylinder *)

	bStateToolDiameter:BYTE;

	(* Max ToolLength *)
	rConvertMaxToolLength:REAL;	(* Convert from cm to mm-->it need for the max value for ToolFeed Position *)

(* Machine Configuration *)
	iConfigMachineType:INT;
	iConfigAxisType:INT;
	iConfigVisuNavigation:INT;
	rConfigMaxToolLength:REAL;
	(* 30.11.2010 KFS:	{	*)
	rConfigMaxToolLengthOriginal:REAL;
	(* 30.11.2010 KFS:	}	*)
(* TeachIn ToolRotation *)
	rActualToolRotationSpeed:REAL;
	rNewToolRotationSpeed:REAL;
(* TeachIn ToolFeeder *)
	rActualToolFeederSpeed:REAL;
	rActualToolFeederPosition:REAL;
	rNewToolFeederPosition:REAL;
	rOldToolFeederPosition:REAL;
(* TeachIn GrindFeeder *)
	rActualGrindFeederSpeed:REAL;
	rActualGrindFeederPosition:REAL;
	rNewGrindFeederPosition:REAL;
	rOldGrindFeederPosition:REAL;

(* Firmware Information ToolLeft *)
	T_ToolLeftSoftwareInfo:ST_SOFTWARE_INFO;
(* Firmware Information ToolCenter *)
	T_ToolCenterSoftwareInfo:ST_SOFTWARE_INFO;
(* Firmware Information ToolRight *)
	T_ToolRightSoftwareInfo:ST_SOFTWARE_INFO;
(* Firmware Information ToolFeeder *)
	T_ToolFeederSoftwareInfo:ST_SOFTWARE_INFO;
(* Firmware Information GrindFeeder *)
	T_GrindFeederSoftwareInfo:ST_SOFTWARE_INFO;

(* Max value ToolRotation *)
	rMaxSpeedToolRotation:REAL;

(* Gilt für die Prozedur für das einstellen des Referenzindex der Achse *)
	iWireFeederAngleRefIndex:INT;
	iWireFeederRefIndexState:INT;
END_STRUCT
END_TYPE

(* Data type in QVis *)
TYPE ST_EXCHG_TEACHIN :
STRUCT
	xSlowFastToolRotation:BOOL;
	xSlowFastToolFeed:BOOL;
	xSlowFastGrindFeeder:BOOL;
	iSelectAxisToolRotation:INT;
	iSelectAxisWireFeeder:INT;
	iSelectAxisGrind:INT;
	iSaveToolFeederPos:INT;
	iSaveGrindFeederPos:INT;
	TParam_ToolLeft:ST_EXCHG_PARAM_TEACHIN;
	TParam_ToolCenter:ST_EXCHG_PARAM_TEACHIN;
	TParam_ToolRight:ST_EXCHG_PARAM_TEACHIN;
	TParam_ToolFeeder:ST_EXCHG_PARAM_TEACHIN;
	TParam_GrindFeeder:ST_EXCHG_PARAM_TEACHIN;
	TParam_AxisPosition:ST_EXCHG_PARAM_POSITION;
END_STRUCT
END_TYPE

(* Data type in QVis *)
TYPE ST_EXCHG_TOUCHSCREENBTPANEL :
STRUCT
	iNotMaskTextBt:INT;
	iActivBtLeft:INT;
	iStateBtLeft:INT;
	iActivBtRight:INT;
END_STRUCT
END_TYPE

(* Data type in QVis *)
TYPE ST_EXCHG_TOUCHSCREENNAVPANEL :
STRUCT
	wState:WORD;
	wNotMasktext:WORD;
	wActivBt:WORD;
END_STRUCT
END_TYPE

(* Data type in QVis *)
TYPE ST_EXCHG_VISU :
STRUCT
(* Message structure *)
	T_Message:ST_EXCHG_MESSAGE;
(* Error List Structure *)
	T_MsgErrorEnglish:ST_EXCHG_MESSAGE_ERROR;
	T_MsgErrorDeutsch:ST_EXCHG_MESSAGE_ERROR;
	T_MsgErrorFrancais:ST_EXCHG_MESSAGE_ERROR;
(* Delete Error List *)
	xDeleteErrorList:BOOL;
(* Level structure *)
	T_Level:ST_EXCHG_LEVEL;
(* Variable *)
	iQVisActivNewPage:INT:=0;
	iLoadingStartPage:INT:=1;
	bActivSpecialLayer:BYTE:=0;
	xKey_Enter:BOOL;
	xKey_Escape:BOOL;

	xLoadingProcessDone:BOOL;
	rSWVersion:REAL:=4500306;	(* V4500306.pro *)

END_STRUCT
END_TYPE

(* Data type in QVis *)
TYPE ST_PAGE :
STRUCT
	iIndexConfigPage:INT:=0;
END_STRUCT
END_TYPE

(* Data type in QVis *)
TYPE ST_QVIS :
STRUCT
	T_PageIndex:ARRAY[1..999] OF ST_PAGE;
	T_ConfigPage:ARRAY[1..csiMaxPage] OF ST_CONFIGPAGE;
	T_CtrleVisu:ST_CTRLEVISU;
	T_PlcParam:ST_VISU_PLC_PARAM;
	T_CtrleAction:ST_CTRLEACTION;
	T_CtrleProcess:ST_CTRLEPROCESS;
	ptrT_ExchgParam:POINTER TO ST_QVIS_EXCHG_PARAM;
END_STRUCT
END_TYPE

(* Data type in QVis *)
TYPE ST_QVIS_EXCHG_PARAM :
STRUCT
	T_Config:ST_EXCHG_CONFIG;
	T_Visu:ST_EXCHG_VISU;
	T_TouchScreenBtPanel:ST_EXCHG_TOUCHSCREENBTPANEL;
	T_BtFunctionPanel:ST_EXCHG_BTFUNCTIONPANEL;
	T_TouchScreenNavPanel:ST_EXCHG_TOUCHSCREENNAVPANEL;
	T_SafetyCtrl:ST_EXCHG_SAFETY_CTRL;

	T_Machine:ST_EXCHG_MACHINE;

	T_TeachIn:ST_EXCHG_TEACHIN;

	T_Cylinder:ST_EXCHG_CYLINDER;

	T_GeometryCommon:ST_GEOMETRY_COMMON;
	T_ProfileCommon:ST_EXCHG_PROFILE_COMMON;
	T_StationCommon:ST_EXCHG_STATION_COMMON;
	T_FunctionCommon:ST_EXCHG_FUNCTION_COMMON;
	T_InfoValueCommon:ST_EXCHG_INFOVALUE_COMMON;

	T_TimeStamp:TIMESTRUCT; (* SOA 12.01.2023*)
END_STRUCT
END_TYPE

(* Data type in QVis *)
TYPE ST_QVISCTRLE :
STRUCT
	dwInCommand:DWORD;
	dwInCount:DWORD;
	dwInQVisCtrlAddress:DWORD;
	dwInParameterAddress:DWORD;
	dwOutCount:DWORD;
	diOutStatus:DINT;
END_STRUCT
END_TYPE

(* Data type in QVis *)
TYPE ST_VISU_PLC_PARAM :
STRUCT
	dwSetNewPage:DWORD;
	dwActualPage:DWORD;
	dwPreviousPage:DWORD;
END_STRUCT
END_TYPE

(* Data type in Retain *)
TYPE ST_CTRLE_DATA_RETAIN :
STRUCT
(* input *)
	xExecute:BOOL:=FALSE;
	xReset:BOOL:=FALSE;
	iFunction:INT:=0;
	udiSrcLen:UDINT;
	udiDestLen:UDINT;
	udipSrcAddr:UDINT;
	udipDestAddr:UDINT;
	tTimeOut:TIME;
	xBlockReadFirstTime:BOOL;

(* Output *)
	xFirstRead:BOOL:=FALSE;
	xDone:BOOL:=FALSE;
	xErr:BOOL:=FALSE;
	udiErrorID:UDINT:=0;
END_STRUCT
END_TYPE

(* Data type in Retain *)
TYPE ST_DATA_RETAIN :
STRUCT
	T_ProcessImageLoadData:ST_RETAIN_DATA_PROCESSIMAGE;		(* All value for a profile, is the value of the profile *)
	T_ProcessImageData:ST_RETAIN_DATA_PROCESSIMAGE;			(* All value for a profile, is the value of the process image parameter *)
	T_Standard:ST_RETAIN_DATA;							(*  *)
	T_IDProfileStation:ARRAY[1..csiMaxProfile] OF ST_PROFILE_ID;	(* List of saved profil *)
	T_ErrorNrList:ST_RETAIN_ERROR_DATA;					(* List of occured error *)

	(*SOA 12.01.2023 {*)
	TWarmUp_Para			:ST_PARA_WARMUP;
	(*SOA 12.01.2023 }*)
END_STRUCT
END_TYPE

(* Data type in Retain *)
TYPE ST_NOVRAM :
STRUCT
	T_Ctrle:ST_CTRLE_DATA_RETAIN;
	T_Data:ST_DATA_RETAIN;
END_STRUCT
END_TYPE

(* Data type in Retain *)
TYPE ST_RETAIN_DATA :
STRUCT
	T_MachineConfig:ST_EXCHG_PARAM_MACHINE_CONFIG;
	T_TeachINToolLeft:ST_EXCHG_PARAM_TEACHIN;
	T_TeachINToolCenter:ST_EXCHG_PARAM_TEACHIN;
	T_TeachINToolRight:ST_EXCHG_PARAM_TEACHIN;
	T_TeachINToolFeeder:ST_EXCHG_PARAM_TEACHIN;
	T_TeachINGrindFeeder:ST_EXCHG_PARAM_TEACHIN;
	T_Cyl_ToolTension:ST_EXCHG_PARAM_CYL_FORCE;
	T_ToolTensionSystem:ST_EXCHG_PARAM_TOOLTENSIONSYSTEM;
	T_InfoProcess:ST_EXCHG_INFO_PROCESS;
	T_AxisPosition:ST_EXCHG_PARAM_POSITION;
END_STRUCT
END_TYPE

(* Data type in Retain *)
TYPE ST_RETAIN_DATA_PROCESSIMAGE :
STRUCT
	T_GeometryPara:ST_GEOMETRY;
	T_PrismPara:ST_EXCHG_PARAM_PRISM;
	T_ProcessPara:ST_EXCHG_PARAM_PROCESS;
	T_AutoGeometryPara:ST_EXCHG_PARAM_AUTOGEOMETRY;
	T_AutoGroovePara:ST_EXCHG_PARAM_AUTOGROOVE;
	T_CalibrationPara:ST_EXCHG_PARAM_CALIBRATION;
END_STRUCT
END_TYPE

(* Data type in Retain *)
TYPE ST_RETAIN_ERROR_DATA :
STRUCT
	adiErrorListMachine:ARRAY [1..20] OF DINT;
	asErrorTimeStampMachine:ARRAY [1..20] OF STRING(12);
END_STRUCT
END_TYPE

(* Data type in StartUp *)
TYPE ST_CTRLESTARTUP :
STRUCT
(* Input *)
	xExecute:BOOL;
	xReset:BOOL;
	iFunction:INT;
	iMsgNumber:INT;
	xSetSecurityStateON:BOOL;
(* Output *)
	xDone:BOOL;
	xErr:BOOL;
	udiErrorID:UDINT;
END_STRUCT
END_TYPE

(* Data type in StartUp *)
TYPE ST_STARTUP :
STRUCT
	T_Ctrle:ST_CTRLESTARTUP;
	T_State:ST_STARTUPSTATE;
END_STRUCT
END_TYPE

(* Data type in StartUp *)
TYPE ST_STARTUPSTATE :
STRUCT
	xPLCReady:BOOL;
	xCompleted:BOOL;
	xBlockChangeMovementVisu:BOOL;	(* For active message overlay, block the visu *)
	xSecurityCircuitActive:BOOL;	(* TRUE = No Energy-->Circuit is open, FALSE = Energy is on-->Circuit is closed *)
	xBlockVisuNavigation:BOOL;		(* For active movement, block the visu *)
END_STRUCT
END_TYPE

(* Data type in Static_Error_List *)
TYPE ST_ERROR_LIST :
STRUCT
	asErrorListEnglish: ST_LANGUAGE_LIST;
	asErrorListDeutsch: ST_LANGUAGE_LIST;
	asErrorListFrancais: ST_LANGUAGE_LIST;
END_STRUCT
END_TYPE

(* Data type in Static_Error_List *)
TYPE ST_LANGUAGE_LIST :
STRUCT
	T_LanguagList:ARRAY [1..255] OF STRING(100);
END_STRUCT
END_TYPE

(* Data type in Station *)
TYPE ST_CONTROL :
STRUCT
	xActiveStation : BOOL;
	xActiveHardware : BOOL;
	xHardwareConfigError : BOOL;
	iFunctNr : INT :=0;
	xEnable : BOOL := FALSE;
	xSecurityCircuitOn : BOOL := FALSE;
	xSecurityCircuitOff : BOOL := FALSE;
	xStart : BOOL := FALSE;
	xEnd : BOOL := FALSE;
	xStop : BOOL := FALSE;
	xRdy : BOOL := FALSE;
	xError : BOOL := FALSE;
	diErrorNr : DINT :=0;
	xQuitError : BOOL := FALSE;
	wStatus : WORD := 0;
	xAbord : BOOL := FALSE;
	xReferenced : BOOL := FALSE;
	xResetReference : BOOL :=FALSE;
	xSetReference : BOOL :=FALSE;
	xHWAxesActive : BOOL := FALSE;
	xActiveMovement : BOOL;
	xResetHardware:BOOL;
	iCountDownPlungeCycle:INT;
END_STRUCT
END_TYPE

(* Data type in Station *)
TYPE ST_CTRL_FUNCTION :
STRUCT
	xStart: BOOL := FALSE;
	xStop: BOOL := FALSE;
	xQuitErr : BOOL := FALSE;
	xStepByStep : BOOL := FALSE;
	xAbord : BOOL := FALSE;
	xEnd : BOOL := FALSE;
	xError : BOOL := FALSE;
	iErrorNr : DINT := 0;
	xReset:BOOL:=FALSE;
END_STRUCT
END_TYPE

(* Data type in Station *)
TYPE ST_HARDWARE :
STRUCT
	TAxisToolLeft:ST_AXIS;
	TAxisToolCenter:ST_AXIS;
	TAxisToolRight:ST_AXIS;
	TAxisToolFeeder:ST_AXIS;
	TAxisGrindFeeder:ST_AXIS;
	TCylToolTension:ST_CYLINDER;
(*22.12.2009: KFS {    *)
	TCylToolLeftActive:ST_CYLINDER;
	TCylToolRightActive:ST_CYLINDER;
	TCylToolCenterActive:ST_CYLINDER;
	TCylToolPrismaLeftActive:ST_CYLINDER;
	TCylToolPrismaRightActive:ST_CYLINDER;
	TToolFeederWorkLength:ST_CYLINDER;
(*22.12.2009: KFS }   *)
END_STRUCT
END_TYPE

(* Data type in Station *)
TYPE ST_STATION :
STRUCT
	xActive : BOOL;
	TControl:ST_CONTROL;
	TCtrlFunction:ST_CTRL_FUNCTION;
	T_WorkTool:ST_WORKTOOL;
	THardware:ST_HARDWARE;
	T_MachineConfig:ST_EXCHG_PARAM_MACHINE_CONFIG;
	rStartPosAutoGrooveToolRotation:REAL;
	xOverwriteMaxToolLength:BOOL;
END_STRUCT
END_TYPE

(* Data type in Station *)
TYPE ST_WORKTOOL :
STRUCT
(* Input parameter *)
	rToolRotationSpeed:REAL;		(* U/Min *)
	rPitch:REAL;						(* mm/U *)
	rToolLength:REAL;				(* cm *)
	rGrindFeederPlunge:REAL;			(* um *)
	iBaseGearDivider:INT;				(* No Unit *)
	rPrismaFactor:REAL;				(* No Unit *)
	rToolRightGearRatio:REAL;			(* No Unit *)
	rToolFeederGearRatio:REAL;		(* No Unit *)
	rToolFeederScaleFactor:REAL;		(* inc/mm *)
	rGrindFeederScaleFactor:REAL;		(* inc/um *)
	rPlungeLengthToolFeed:REAL;		(* mm *)
	rPlungeSpeedGrindFeed:REAL;		(* um/s *)
	rDisplaceLengthToolFeed:REAL;	(* mm *)
	rDisplaceSpeedGrindFeed:REAL;	(* um/s *)
	xPlungeActivation:BOOL;			(* No Unit *)
	xDisplaceActivation:BOOL;			(* No Unit *)
(* Output parameter *)
	rToolRotationSpeedMotor:REAL;	(* inc/64s *)
	rToolFeederSpeedUnit:REAL;		(* mm/s *)
	rToolFeederSpeedMotorRel:REAL;	(* inc/64s *)
	rToolFeederSpeedMotorAbs:REAL;	(* inc/64s *)
	iToolFeederGearFactor:INT;		(* No Unit *)
	iToolFeederGearDivider:INT;		(* No Unit *)
	rToolFeederRelPositionUnit:REAL;	(* mm *)
	rToolFeederRelPositionMotor:REAL;	(* inc *)
	rGrindFeederSpeedUnit:REAL;		(* um/s *)
	rGrindFeederSpeedMotor:REAL;	(* inc/um *)
	rTimeLeftWork:REAL;				(* s *)
	iTotalCountDownPlungeCycle:INT;	(* No Unit *)
END_STRUCT
END_TYPE

(* Data type in TwinSAFE *)
TYPE ST_TWINSAFE_CTRLE_IN :
STRUCT
	xTwinSAFE_Group_FB_Error: BOOL;
	xTwinSAFE_Group_COM_Error: BOOL;
	xTwinSAFE_Group_OUT_Error: BOOL;
END_STRUCT
END_TYPE

(* Data type in TwinSAFE *)
TYPE ST_TWINSAFE_CTRLE_OUT :
STRUCT
	xTwinSAFE_Run: BOOL;
	xTwinSAFE_Reset: BOOL;
END_STRUCT
END_TYPE

(* Data type in TwinSAFE *)
TYPE ST_TWINSAFE_IN :
STRUCT
(* KL1904, Input *)
	IxReadyToolLeft:BOOL;
	IxReadyToolCenter:BOOL;
	IxReadyToolRight:BOOL;
	IxReadyToolFeeder:BOOL;
	IxReadyGrindFeeder:BOOL;
	IxRealseButton:BOOL;
	IxEmergencyStopStuder:BOOL;
	IxEmergencyStopMachine:BOOL;
	IxPowerSupplyEcoStep:BOOL;
	IxContactorAuxContact:BOOL;
END_STRUCT
END_TYPE

(* Data type in TwinSAFE *)
TYPE ST_TWINSAFE_OUT :
STRUCT
(* KL6904, Output *)
	QxEmergencyStopStuder:BOOL;
	QxAirSupply:BOOL;
	QxContactor_K3:BOOL;
	QxContactor_K4:BOOL;
END_STRUCT
END_TYPE

(* POU PRG_STARTUP, ST *)
PROGRAM PRG_STARTUP
VAR
	xRdy: BOOL;
	iStepAction: INT := 10;
	xFirstExecution: BOOL;
	xPLCWait: BOOL := TRUE;
	TONPLCWait: TON;
	tTimeOutFunction: TIME;
	TimerFunction: TON;
	RisingEdgeExecute: R_TRIG;
	xInitVisu: BOOL;
	xLoading: BOOL;
	TONStartUp: TON;
	xReboot: BOOL;
	xEmergency: BOOL;
	xStartBooting: BOOL;
	xNoAirPressure: BOOL;
	xNodeFailCANOpen: BOOL;
	xActiveErrorMsg: BOOL;
	iMsgNumber: INT;
	xActiveInfoMsg: BOOL;
	iStepFunction: INT;
	RisingEdgeQuitButton: R_TRIG;
	RisingEdgeStartButton: R_TRIG;
	TONWaitResetOutput: TON;
	xStartCheck: BOOL:=TRUE;
	xDeleteErrorMessage: BOOL;
	TONWaitCircuitOn: TON;
	xCheckSecurityDoor: BOOL;
	tTimeStartUp: TIME := T#120ms;
	TimerDelayStartStation: TON;
	xTmp: BOOL;
	xReadHardware: BOOL;
	xTmp1: BOOL;
	xCheckConfirm: BOOL;
(* variable *)
(* Execute *)
	xSetOutputDisable:BOOL;
(* Init Error List *)
	FallingEdgeSecurityCircuit1:F_TRIG;
	FallingEdgeSecurityCircuit2:F_TRIG;
	RisingEdgeSecurityCircuit1:R_TRIG;
	RisingEdgeSecurityCircuit2:R_TRIG;
	FallingEdgeEnergyOff:F_TRIG;
	RisingEdgeEnergyOn:R_TRIG;
	TONWaitEndMessage:TON;
	xCheckAirPressure: BOOL;
	TONWaitCheckAirPressure: TON;
	xSwitchOffMachine: BOOL;
	TONWaitSwitchOffMachine: TON;
	iStepSwitchOffMachine: INT;
	xSwitchOffMachineReady: BOOL;
	xBlockChecking: BOOL;
	xCheckStateSecurityDoor: BOOL;
	xProcessAbordet: BOOL;
(* Init Error List *)
	FBInitErrorList:FB_InitErrorList;
	FBBIOSPARAMETER: FB_BIOSPARAMETER;
	FBErrorMessage : FB_ErrorMessage;
	diTmpErrorNr: DINT;
	FBCheckActiveMovement: FB_CHECKACTIVEMOVEMENT;
	xResetFBActiveMovement: BOOL;
	RisingEdgeTemp: R_TRIG;
	xTmpSecurityKey: BOOL;
	xMicroRodActive: BOOL;
	iStepFunctionON: INT;
	xReadFirstTime: BOOL;
	TONWaitSetSecStateON: TON;
	xCheckStateOfDrive: BOOL;
	TONChkStateDrive: TON;
	xSwitchOffHardwareLayer: BOOL;
	xTmp2: BOOL;
END_VAR
(****************************************************************************************************************************************************)
(**********      This Functionblock manage the booting of the machine and the security mangament of the machine during   ********)
(**********       the machine operating                           														    ************)
(****************************************************************************************************************************************************)
(* First execution of the start up *)
IF NOT(xFirstExecution) THEN
	(* Init. Startup structure *)
	T_StartUp.T_Ctrle.xExecute:=FALSE;
	T_StartUp.T_Ctrle.xDone:=FALSE;
	T_StartUp.T_Ctrle.xErr:=FALSE;
	T_StartUp.T_Ctrle.xReset:=FALSE;
	T_StartUp.T_State.xPLCReady:=FALSE;
	T_StartUp.T_Ctrle.iFunction:=0;
	T_StartUp.T_Ctrle.udiErrorID:=16#0;
	T_StartUp.T_State.xBlockChangeMovementVisu:=TRUE;
	T_StartUp.T_Ctrle.iMsgNumber:=0;
	(* Timer *)
	TimerFunction(IN:=FALSE);
	(* confirm first execution *)
	xFirstExecution:=TRUE;
	TONPLCWait(IN:=FALSE);
	RETURN;
END_IF

(* waiting 5 sec before starting *)
	IF xPLCWait THEN
		TONPLCWait(IN:=TRUE,PT:=T#5s);
		IF TONPLCWait.Q THEN
			TONPLCWait(IN:=FALSE);
			xPLCWait:=FALSE;
			(* activ function "Start PLC" *)
			T_StartUp.T_Ctrle.xExecute:=TRUE;
			T_StartUp.T_Ctrle.iFunction:=1;
			tTimeOutFunction:=T#2s;
		END_IF;
		RETURN;
	END_IF;

(****************************************************************************************************************************************************)
(***********                                start of the check for the emergeny button, air and axis communication error                              ************)
(****************************************************************************************************************************************************)
(* check the emergency stop and the air pressure after booting the machine *)
	IF NOT(xStartCheck) THEN
	(* check emergency stop, only if it is not already in this state *)
		IF NOT(xStartBooting AND ((iStepFunction = 1) OR (iStepFunction = 10))) THEN
			IF NOT(T_TwinSafeIn.IxEmergencyStopMachine) OR NOT(T_TwinSafeIn.IxEmergencyStopStuder) THEN
				IF NOT((xEmergency AND (iStepFunction < 40))) THEN
					RisingEdgeExecute(CLK:=FALSE);
					(* Set emergency function *)
					T_StartUp.T_Ctrle.xExecute:=TRUE;
					T_StartUp.T_Ctrle.iFunction:=4;
					xInitVisu:=FALSE;
					xLoading:=FALSE;
					xReboot:=FALSE;
					xStartBooting:=FALSE;
					xActiveErrorMsg:=FALSE;
					xActiveInfoMsg:=FALSE;
					xCheckConfirm:=FALSE;
					xSwitchOffMachineReady:=FALSE;
					xSwitchOffMachine:=FALSE;
					xNoAirPressure:=FALSE;
					xNodeFailCANOpen:=FALSE;
					xResetFBActiveMovement:=TRUE;
					tTimeOutFunction:=T#0s;
					T_StartUp.T_State.xCompleted:=FALSE;
				END_IF;
			END_IF;
		END_IF;
	
	(* check air pressure, only if it is not already in this state *)
		IF NOT(xStartBooting) AND NOT(xEmergency) THEN
			IF T_TwinSafeIn.IxEmergencyStopMachine AND T_TwinSafeIn.IxEmergencyStopStuder AND NOT(IarxDigitalInput[4]) THEN
				IF T_TwinSafeOut.QxContactor_K3 AND T_TwinSafeOut.QxContactor_K4 AND NOT(xNoAirPressure) THEN
					xCheckAirPressure:=TRUE;
				END_IF;
			ELSE
				TONWaitCheckAirPressure(IN:=FALSE);
				xCheckAirPressure:=FALSE;
			END_IF;
			IF xCheckAirPressure THEN
				TONWaitCheckAirPressure(IN:=TRUE,PT:=T#2s);
				IF TONWaitCheckAirPressure.Q THEN
					xCheckAirPressure:=FALSE;
					TONWaitCheckAirPressure(IN:=FALSE);
					IF NOT(IarxDigitalInput[4]) THEN
						RisingEdgeExecute(CLK:=FALSE);
						(* Set No Air pressure function *)
						T_StartUp.T_Ctrle.xExecute:=TRUE;
						T_StartUp.T_Ctrle.iFunction:=6;
						xInitVisu:=FALSE;
						xLoading:=FALSE;
						xReboot:=FALSE;
						xStartBooting:=FALSE;
						xActiveErrorMsg:=FALSE;
						xActiveInfoMsg:=FALSE;
						xCheckConfirm:=FALSE;
						xCheckSecurityDoor:=FALSE;
						xCheckStateSecurityDoor:=FALSE;
						xSwitchOffMachineReady:=FALSE;
						xSwitchOffMachine:=FALSE;
						xResetFBActiveMovement:=TRUE;
						tTimeOutFunction:=T#0s;
						T_StartUp.T_State.xCompleted:=FALSE;
					END_IF;
				END_IF;
			END_IF;
		ELSE
			xCheckAirPressure:=FALSE;
			TONWaitCheckAirPressure(IN:=FALSE);
		END_IF;
	END_IF;

	(* check Node of the Ventilinsel, only if it is not already in this state *)
	IF NOT(xStartBooting) AND NOT(xEmergency) AND NOT(xCheckAirPressure) AND T_StartUp.T_State.xCompleted AND NOT(xNoAirPressure) AND NOT(xNodeFailCANOpen) THEN
		xTmp:=	(T_AxisNodeState.bToolLeftNodeState <> 0) OR
				((T_AxisNodeState.bToolCenterNodeState <> 0) AND xMicroRodActive) OR
				(T_AxisNodeState.bToolRightNodeState <> 0) OR
				(T_AxisNodeState.bToolFeederNodeState <> 0) OR
				(T_AxisNodeState.bGrindFeederNodeState <> 0);
		IF xTmp THEN
			RisingEdgeExecute(CLK:=FALSE);
			(* Set CANOpen NodeFail function *)
			T_StartUp.T_Ctrle.xExecute:=TRUE;
			T_StartUp.T_Ctrle.iFunction:=7;
			xInitVisu:=FALSE;
			xLoading:=FALSE;
			xReboot:=FALSE;
			xStartBooting:=FALSE;
			xActiveErrorMsg:=FALSE;
			xActiveInfoMsg:=FALSE;
			xCheckConfirm:=FALSE;
			xCheckSecurityDoor:=FALSE;
			xCheckStateSecurityDoor:=FALSE;
			xSwitchOffMachineReady:=FALSE;
			xSwitchOffMachine:=FALSE;
			xResetFBActiveMovement:=TRUE;
			tTimeOutFunction:=T#0s;
			T_StartUp.T_State.xCompleted:=FALSE;
		END_IF;
	END_IF;
(****************************************************************************************************************************************************)
(***********                                end of the check for the emergeny button, air and axis communication error                              ************)
(****************************************************************************************************************************************************)

(****************************************************************************************************************************************************)
(***********                                               start of the management for calling of the start up function                                                   ************)
(****************************************************************************************************************************************************)
(* execute *)
	RisingEdgeExecute(CLK:=T_StartUp.T_Ctrle.xExecute);
	T_StartUp.T_Ctrle.xExecute:=FALSE;
	IF RisingEdgeExecute.Q THEN
		T_StartUp.T_Ctrle.xExecute:=FALSE;
		CASE T_StartUp.T_Ctrle.iFunction OF
		(* Start PLC *)
		1:	xInitVisu:=TRUE;
			tTimeOutFunction:=T#2s;
		(* Start loading *)
		2:	xLoading:=TRUE;
			T_VisuQVis.ptrT_ExchgParam^.T_Visu.iLoadingStartPage:=1;
			tTimeOutFunction:=T#60s;
			TONStartUp(IN:=FALSE);
		(* Start reboot *)
		3:	xReboot:=TRUE;
			tTimeOutFunction:=T#5s;
		(* Emergency *)
		4:	xEmergency:=TRUE;
			tTimeOutFunction:=T#0s;	(* No Time out *)
		(* Start Booting *)
		5:	xStartBooting:=TRUE;
			tTimeOutFunction:=T#0s;	(* No Time out *)
		(* No Air pressure *)
		6:	xNoAirPressure:=TRUE;
			tTimeOutFunction:=T#0s;	(* No Time out *)
		(* Node CANOpen fail *)
		7:	xNodeFailCANOpen:=TRUE;
			tTimeOutFunction:=T#0s;	(* No Time out *)
		(* Read NovRAM Parameter *)
		8:	xReadHardware:=TRUE;
			tTimeOutFunction:=T#5s;
		(* Activate Error Message Overlay *)
		10:	xActiveErrorMsg:=TRUE;
			iMsgNumber:=T_StartUp.T_Ctrle.iMsgNumber;
			T_StartUp.T_Ctrle.iMsgNumber:=0;
			tTimeOutFunction:=T#0s;	(* No Time out *)
			T_StartUp.T_State.xBlockChangeMovementVisu:=TRUE;	(* Lock the navigation of the visu *)
		(* Acitvate Info Message Overlay *)
		11:	xActiveInfoMsg:=TRUE;
			iMsgNumber:=T_StartUp.T_Ctrle.iMsgNumber;
			T_StartUp.T_Ctrle.iMsgNumber:=0;
			tTimeOutFunction:=T#0s;	(* No Time out *)
			T_StartUp.T_State.xBlockChangeMovementVisu:=TRUE;	(* Lock the navigation of the visu *)
		ELSE
		(* function not implemented *)
			T_StartUp.T_Ctrle.xDone:=FALSE;
			T_StartUp.T_Ctrle.xErr:=TRUE;
			T_StartUp.T_Ctrle.udiErrorID:=16#F000;
			(* Exit FB *)
			RETURN;
		END_CASE
		(* Init. variable *)
		iStepFunction:=1;
		T_StartUp.T_Ctrle.xDone:=FALSE;
		T_StartUp.T_Ctrle.xErr:=FALSE;
		T_StartUp.T_Ctrle.udiErrorID:=0;
		TimerFunction(IN:=FALSE);
	(* Exit FB *)
		RETURN;
	END_IF
(****************************************************************************************************************************************************)
(***********                                               end of the management for calling of the start up function                                                   ************)
(****************************************************************************************************************************************************)

(* Start and Quit Button *)
	RisingEdgeStartButton(CLK:=IarxDigitalInput[1]);
	RisingEdgeQuitButton(CLK:=T_TwinSafeIn.IxRealseButton);

(* Check of the failed function for the drive. If an error exist on the Axis and the current is off, than it gives not a possibility to switch on the energy. This part will check this state and reset the error *)
	IF (NOT(T_TwinSafeOut.QxContactor_K3) OR NOT(T_TwinSafeOut.QxContactor_K4)) THEN
		IF RisingEdgeQuitButton.Q THEN
			xCheckStateOfDrive:=TRUE;
			TONChkStateDrive(IN:=FALSE);
		END_IF;
		IF xCheckStateOfDrive THEN
			TONChkStateDrive(IN:=TRUE,PT:=T#2s);
			IF TONChkStateDrive.Q THEN
				xCheckStateOfDrive:=FALSE;
				IF NOT(T_Station.TControl.xActiveHardware) THEN
					xSwitchOffHardwareLayer:=TRUE;
					T_Station.TControl.xActiveHardware:=TRUE;
				END_IF;
				IF T_TwinSafeIn.IxReadyToolLeft AND T_Station.THardware.TAxisToolLeft.T_CtrleSingle.xErr AND
				     NOT(T_Station.THardware.TAxisToolLeft.T_CtrleSingle.xDone) AND NOT(T_Station.THardware.TAxisToolLeft.T_CtrleSingle.xExecute) THEN
					T_Station.THardware.TAxisToolLeft.T_CtrleSingle.iFunction:=1;
					T_Station.THardware.TAxisToolLeft.T_CtrleSingle.xExecute:=TRUE;
				END_IF;
				IF xMicroRodActive THEN
					IF T_TwinSafeIn.IxReadyToolCenter AND T_Station.THardware.TAxisToolCenter.T_CtrleSingle.xErr AND
					     NOT(T_Station.THardware.TAxisToolCenter.T_CtrleSingle.xDone) AND NOT(T_Station.THardware.TAxisToolCenter.T_CtrleSingle.xExecute) THEN
						T_Station.THardware.TAxisToolCenter.T_CtrleSingle.iFunction:=1;
						T_Station.THardware.TAxisToolCenter.T_CtrleSingle.xExecute:=TRUE;
					END_IF;
				END_IF;
				IF T_TwinSafeIn.IxReadyToolRight AND T_Station.THardware.TAxisToolRight.T_CtrleSingle.xErr AND
				     NOT(T_Station.THardware.TAxisToolRight.T_CtrleSingle.xDone) AND NOT(T_Station.THardware.TAxisToolRight.T_CtrleSingle.xExecute) THEN
					T_Station.THardware.TAxisToolRight.T_CtrleSingle.iFunction:=1;
					T_Station.THardware.TAxisToolRight.T_CtrleSingle.xExecute:=TRUE;
				END_IF;
				IF T_TwinSafeIn.IxReadyToolFeeder AND T_Station.THardware.TAxisToolFeeder.T_CtrleSingle.xErr AND
				     NOT(T_Station.THardware.TAxisToolFeeder.T_CtrleSingle.xDone) AND NOT(T_Station.THardware.TAxisToolFeeder.T_CtrleSingle.xExecute) THEN
					T_Station.THardware.TAxisToolFeeder.T_CtrleSingle.iFunction:=1;
					T_Station.THardware.TAxisToolFeeder.T_CtrleSingle.xExecute:=TRUE;
				END_IF;
				IF T_TwinSafeIn.IxReadyGrindFeeder AND T_Station.THardware.TAxisGrindFeeder.T_CtrleSingle.xErr AND
				     NOT(T_Station.THardware.TAxisGrindFeeder.T_CtrleSingle.xDone) AND NOT(T_Station.THardware.TAxisGrindFeeder.T_CtrleSingle.xExecute) THEN
					T_Station.THardware.TAxisGrindFeeder.T_CtrleSingle.iFunction:=1;
					T_Station.THardware.TAxisGrindFeeder.T_CtrleSingle.xExecute:=TRUE;
				END_IF;
			END_IF;
		END_IF;
	ELSE
		xCheckStateOfDrive:=FALSE;
		TONChkStateDrive(IN:=FALSE);
	END_IF;
	IF xSwitchOffHardwareLayer THEN
		xTmp2:=	T_Station.THardware.TAxisToolLeft.T_CtrleSingle.xDone AND ((T_Station.THardware.TAxisToolCenter.T_CtrleSingle.xDone AND xMicroRodActive) OR NOT(xMicroRodActive)) AND
				T_Station.THardware.TAxisToolRight.T_CtrleSingle.xDone AND T_Station.THardware.TAxisToolFeeder.T_CtrleSingle.xDone AND
				T_Station.THardware.TAxisGrindFeeder.T_CtrleSingle.xDone;
		IF xTmp2 THEN
			xSwitchOffHardwareLayer:=FALSE;
			T_Station.TControl.xActiveHardware:=FALSE;
		END_IF;
	END_IF;

(* Time out function *)
	IF tTimeOutFunction <> T#0s THEN TimerFunction(IN:=TRUE,PT:=tTimeOutFunction); ELSE TimerFunction(IN:=FALSE); END_IF
	IF TimerFunction.Q AND NOT T_StartUp.T_Ctrle.xDone AND NOT T_StartUp.T_Ctrle.xErr THEN
	(* Error, timeout action activ *)
		T_StartUp.T_Ctrle.xErr:=TRUE;
		(* Init. variable *)
		xInitVisu:=FALSE;
		xLoading:=FALSE;
		xReboot:=FALSE;
		xStartBooting:=FALSE;
		xActiveErrorMsg:=FALSE;
		xActiveInfoMsg:=FALSE;
		xCheckSecurityDoor:=FALSE;
		xCheckStateSecurityDoor:=FALSE;
		(* Set output disable *)
		xSetOutputDisable:=TRUE;
		(* Display error message *)
		T_VisuQVis.ptrT_ExchgParam^.T_Visu.T_Message.iState:=203;
		(* exit FB, do not continue the execution of action! *)
		(* Overlay Message Error *)
		T_VisuQVis.ptrT_ExchgParam^.T_SafetyCtrl.bStateMessageError:=1;
		T_VisuQVis.ptrT_ExchgParam^.T_SafetyCtrl.bStateMessageInfo:=0;
		T_VisuQVis.ptrT_ExchgParam^.T_SafetyCtrl.bStateMessageWarning:=0;
		T_VisuQVis.ptrT_ExchgParam^.T_SafetyCtrl.iMsgErrorLine1:=7;	(* WHILE THE MACHINE IS BOOTING *)
		T_VisuQVis.ptrT_ExchgParam^.T_SafetyCtrl.iMsgErrorLine2:=7;	(* AN ERROR IS OCCURRED *)
		T_VisuQVis.ptrT_ExchgParam^.T_SafetyCtrl.iMsgErrorLine3:=7;	(* PLEASE CONFIRM THIS MESSAGE AND READ AFTER *)
		T_VisuQVis.ptrT_ExchgParam^.T_SafetyCtrl.iMsgErrorLine4:=7;	(* THE ACCORDING ERROR *)
		T_VisuQVis.ptrT_ExchgParam^.T_SafetyCtrl.xConfirmMsgError:=FALSE;
		T_VisuQVis.ptrT_ExchgParam^.T_SafetyCtrl.xBlockVisuObject:=TRUE;
		xCheckConfirm:=TRUE;
	END_IF
	IF xCheckConfirm AND NOT(xEmergency) AND NOT(xNoAirPressure) AND NOT(xNodeFailCANOpen) THEN
		IF T_VisuQVis.ptrT_ExchgParam^.T_SafetyCtrl.xConfirmMsgError THEN
			T_VisuQVis.ptrT_ExchgParam^.T_SafetyCtrl.xBlockVisuObject:=FALSE;
			T_VisuQVis.ptrT_ExchgParam^.T_SafetyCtrl.bStateMessageError:=0;
			T_VisuQVis.ptrT_ExchgParam^.T_SafetyCtrl.xConfirmMsgError:=FALSE;
			xCheckConfirm:=FALSE;
			xStartBooting:=TRUE;
			tTimeOutFunction:=T#0s;	(* deactivate the time out *)
			(* next step *)
			iStepFunction:=1;
		END_IF;
	ELSE
		xCheckConfirm:=FALSE;
	END_IF;

(* Check Lamp State of external Button *)
	IF NOT(T_StartUp.T_State.xCompleted) THEN
		IF (NOT(T_TwinSafeOut.QxContactor_K3) OR NOT(T_TwinSafeOut.QxContactor_K4)) THEN
			QarxDigitalOutput[1]:=FALSE;
			QarxDigitalOutput[2]:=FALSE;
			QarxDigitalOutput[3]:=TRUE;
		END_IF;
		IF T_TwinSafeOut.QxContactor_K3 AND T_TwinSafeOut.QxContactor_K4 THEN
			QarxDigitalOutput[3]:=FALSE;
		END_IF;
		IF NOT(T_TwinSafeIn.IxPowerSupplyEcoStep) THEN
			QarxDigitalOutput[3]:=FALSE;
		END_IF;
		IF (T_VisuQVis.ptrT_ExchgParam^.T_SafetyCtrl.bStateMessageError <> 0) THEN
			QarxDigitalOutput[1]:=FALSE;
			QarxDigitalOutput[2]:=FALSE;
			QarxDigitalOutput[3]:=FALSE;
		END_IF;
	ELSE
		IF NOT(T_TwinSafeIn.IxPowerSupplyEcoStep) THEN
			QarxDigitalOutput[3]:=FALSE;
		END_IF;
		IF T_TwinSafeIn.IxPowerSupplyEcoStep AND (NOT(T_TwinSafeOut.QxContactor_K3) OR NOT(T_TwinSafeOut.QxContactor_K4)) THEN
			QarxDigitalOutput[3]:=TRUE;
		END_IF;
	END_IF;

(* Check Machine active movement *)
	FBCheckActiveMovement(	T_TwinSafeOut:= T_TwinSafeOut,
							xKeySwitch:= IarxDigitalInput[3],
							xBlockChecking:= xBlockChecking,
							xReset:= xResetFBActiveMovement,
							T_Visu:= T_VisuQVis,
							T_Station:= T_Station,
							T_Process:= T_Process);

(* Message Energy on/off *)
	FallingEdgeEnergyOff(CLK:=NOT(T_TwinSafeOut.QxContactor_K3 AND T_TwinSafeOut.QxContactor_K4));
	RisingEdgeEnergyOn(CLK:=NOT(T_TwinSafeOut.QxContactor_K3 AND T_TwinSafeOut.QxContactor_K4));
	IF T_StartUp.T_State.xCompleted AND FallingEdgeEnergyOff.Q AND NOT(xCheckStateSecurityDoor) THEN
		IF (T_VisuQVis.ptrT_ExchgParam^.T_Visu.T_Message.iState = 0) OR (T_VisuQVis.ptrT_ExchgParam^.T_Visu.T_Message.iState = 119) THEN
			T_VisuQVis.ptrT_ExchgParam^.T_Visu.T_Message.iState:=118;	(* The energy supply is ON *)
			TONWaitEndMessage(IN:=FALSE);
		END_IF;
	END_IF;
	IF T_StartUp.T_State.xCompleted AND RisingEdgeEnergyOn.Q AND NOT(xCheckStateSecurityDoor) THEN
		IF (T_VisuQVis.ptrT_ExchgParam^.T_Visu.T_Message.iState = 0) OR (T_VisuQVis.ptrT_ExchgParam^.T_Visu.T_Message.iState = 118) THEN
			T_VisuQVis.ptrT_ExchgParam^.T_Visu.T_Message.iState:=119;	(* The energy supply is OFF *)
			TONWaitEndMessage(IN:=FALSE);
		END_IF;
	END_IF;
	IF (T_VisuQVis.ptrT_ExchgParam^.T_Visu.T_Message.iState = 118) OR (T_VisuQVis.ptrT_ExchgParam^.T_Visu.T_Message.iState = 119) THEN
		TONWaitEndMessage(IN:=TRUE,PT:=T#2s);
		IF TONWaitEndMessage.Q THEN
			TONWaitEndMessage(IN:=FALSE);
			T_VisuQVis.ptrT_ExchgParam^.T_Visu.T_Message.iState:=0;	(* Close Message *)
		END_IF;
	END_IF;

(* Check Power switch off from the security circuit *)
	FallingEdgeSecurityCircuit1(CLK:=T_TwinSafeOut.QxContactor_K3);
	FallingEdgeSecurityCircuit2(CLK:=T_TwinSafeOut.QxContactor_K4);
	IF T_StartUp.T_State.xCompleted AND (FallingEdgeSecurityCircuit1.Q OR FallingEdgeSecurityCircuit2.Q) THEN
		IF (T_VisuQVis.ptrT_ExchgParam^.T_Visu.T_Message.iState <> 401) THEN
			T_VisuQVis.ptrT_ExchgParam^.T_SafetyCtrl.bStateAutoGeometry:=3;
			T_VisuQVis.ptrT_ExchgParam^.T_SafetyCtrl.bStateAutoGroove:=3;
			T_VisuQVis.ptrT_ExchgParam^.T_SafetyCtrl.bStateReference:=3;
			T_VisuQVis.ptrT_ExchgParam^.T_SafetyCtrl.bStateToolCalibration:=3;
			T_VisuQVis.ptrT_ExchgParam^.T_SafetyCtrl.bStateToolTorque:=3;
			T_VisuQVis.ptrT_ExchgParam^.T_SafetyCtrl.bStateTeachInToolLeft:=3;
			T_VisuQVis.ptrT_ExchgParam^.T_SafetyCtrl.bStateTeachInToolCenter:=3;
			T_VisuQVis.ptrT_ExchgParam^.T_SafetyCtrl.bStateTeachInToolRight:=3;
			T_VisuQVis.ptrT_ExchgParam^.T_SafetyCtrl.bStateTeachInToolFeeder:=3;
			T_VisuQVis.ptrT_ExchgParam^.T_SafetyCtrl.bStateTeachInGrindFeeder:=3;
			T_VisuQVis.ptrT_ExchgParam^.T_StationCommon.iWireFeederRefIndexState:=3;
		END_IF;
		IF T_Station.TControl.xActiveHardware THEN
			T_Station.TControl.xSecurityCircuitOff:=TRUE;
			T_Station.TControl.xSecurityCircuitOn:=FALSE;
		END_IF;
		IF T_Process.xEnable AND NOT(T_Process.xEnd) AND ((T_Process.iFunctNr = 10) OR (T_Process.iFunctNr = 20) OR (T_Process.iFunctNr = 30) OR (T_Process.iFunctNr = 40)) THEN
			T_StartUp.T_State.xBlockChangeMovementVisu:=FALSE;
			xProcessAbordet:=TRUE;
		ELSE
			xProcessAbordet:=FALSE;
		END_IF;
		IF NOT(T_Process.xError) THEN
			T_Process.xEnable:=FALSE;
		END_IF;
		QarxDigitalOutput[3]:=TRUE;	(* QxCtrlLampReleaseButton *)
		IF FBCheckActiveMovement.xActiveSetupLevel AND (FBCheckActiveMovement.xActiveProcess OR FBCheckActiveMovement.xActiveStation OR FBCheckActiveMovement.xActiveHWStation) THEN
			xBlockChecking:=TRUE;
		ELSE
			xBlockChecking:=FALSE;
		END_IF;
	END_IF;
	IF NOT(T_TwinSafeIn.IxPowerSupplyEcoStep) THEN
		T_VisuQVis.ptrT_ExchgParam^.T_SafetyCtrl.bStateAutoGeometry:=4;
		T_VisuQVis.ptrT_ExchgParam^.T_SafetyCtrl.bStateAutoGroove:=4;
		T_VisuQVis.ptrT_ExchgParam^.T_SafetyCtrl.bStateReference:=4;
		T_VisuQVis.ptrT_ExchgParam^.T_SafetyCtrl.bStateToolCalibration:=4;
		T_VisuQVis.ptrT_ExchgParam^.T_SafetyCtrl.bStateToolTorque:=4;
		T_VisuQVis.ptrT_ExchgParam^.T_SafetyCtrl.bStateTeachInToolLeft:=4;
		T_VisuQVis.ptrT_ExchgParam^.T_SafetyCtrl.bStateTeachInToolCenter:=4;
		T_VisuQVis.ptrT_ExchgParam^.T_SafetyCtrl.bStateTeachInToolRight:=4;
		T_VisuQVis.ptrT_ExchgParam^.T_SafetyCtrl.bStateTeachInToolFeeder:=4;
		T_VisuQVis.ptrT_ExchgParam^.T_SafetyCtrl.bStateTeachInGrindFeeder:=4;
		T_VisuQVis.ptrT_ExchgParam^.T_StationCommon.iWireFeederRefIndexState:=4;
	END_IF;
	IF T_TwinSafeIn.IxPowerSupplyEcoStep AND (NOT(T_TwinSafeOut.QxContactor_K3) OR NOT(T_TwinSafeOut.QxContactor_K4)) THEN
		T_VisuQVis.ptrT_ExchgParam^.T_SafetyCtrl.bStateAutoGeometry:=3;
		T_VisuQVis.ptrT_ExchgParam^.T_SafetyCtrl.bStateAutoGroove:=3;
		T_VisuQVis.ptrT_ExchgParam^.T_SafetyCtrl.bStateReference:=3;
		T_VisuQVis.ptrT_ExchgParam^.T_SafetyCtrl.bStateToolCalibration:=3;
		T_VisuQVis.ptrT_ExchgParam^.T_SafetyCtrl.bStateToolTorque:=3;
		T_VisuQVis.ptrT_ExchgParam^.T_SafetyCtrl.bStateTeachInToolLeft:=3;
		T_VisuQVis.ptrT_ExchgParam^.T_SafetyCtrl.bStateTeachInToolCenter:=3;
		T_VisuQVis.ptrT_ExchgParam^.T_SafetyCtrl.bStateTeachInToolRight:=3;
		T_VisuQVis.ptrT_ExchgParam^.T_SafetyCtrl.bStateTeachInToolFeeder:=3;
		T_VisuQVis.ptrT_ExchgParam^.T_SafetyCtrl.bStateTeachInGrindFeeder:=3;
		T_VisuQVis.ptrT_ExchgParam^.T_StationCommon.iWireFeederRefIndexState:=3;
	END_IF;
	IF (T_VisuQVis.ptrT_ExchgParam^.T_Visu.T_Message.iState = 401) THEN
		T_VisuQVis.ptrT_ExchgParam^.T_SafetyCtrl.bStateAutoGeometry:=0;
		T_VisuQVis.ptrT_ExchgParam^.T_SafetyCtrl.bStateAutoGroove:=0;
		T_VisuQVis.ptrT_ExchgParam^.T_SafetyCtrl.bStateReference:=0;
		T_VisuQVis.ptrT_ExchgParam^.T_SafetyCtrl.bStateToolCalibration:=0;
		T_VisuQVis.ptrT_ExchgParam^.T_SafetyCtrl.bStateToolTorque:=0;
		T_VisuQVis.ptrT_ExchgParam^.T_SafetyCtrl.bStateTeachInToolLeft:=0;
		T_VisuQVis.ptrT_ExchgParam^.T_SafetyCtrl.bStateTeachInToolCenter:=0;
		T_VisuQVis.ptrT_ExchgParam^.T_SafetyCtrl.bStateTeachInToolRight:=0;
		T_VisuQVis.ptrT_ExchgParam^.T_SafetyCtrl.bStateTeachInToolFeeder:=0;
		T_VisuQVis.ptrT_ExchgParam^.T_SafetyCtrl.bStateTeachInGrindFeeder:=0;
		T_VisuQVis.ptrT_ExchgParam^.T_StationCommon.iWireFeederRefIndexState:=0;
	END_IF;

(* Check Power switch on from the security circuit *)
	RisingEdgeSecurityCircuit1(CLK:=T_TwinSafeOut.QxContactor_K3);
	RisingEdgeSecurityCircuit2(CLK:=T_TwinSafeOut.QxContactor_K4);
	IF T_StartUp.T_State.xCompleted AND (RisingEdgeSecurityCircuit1.Q OR RisingEdgeSecurityCircuit2.Q) THEN
		T_VisuQVis.ptrT_ExchgParam^.T_SafetyCtrl.bStateAutoGeometry:=1;
		T_VisuQVis.ptrT_ExchgParam^.T_SafetyCtrl.bStateAutoGroove:=1;
		T_VisuQVis.ptrT_ExchgParam^.T_SafetyCtrl.bStateReference:=1;
		T_VisuQVis.ptrT_ExchgParam^.T_SafetyCtrl.bStateToolCalibration:=1;
		T_VisuQVis.ptrT_ExchgParam^.T_SafetyCtrl.bStateToolTorque:=1;
		T_VisuQVis.ptrT_ExchgParam^.T_SafetyCtrl.bStateTeachInToolLeft:=1;
		T_VisuQVis.ptrT_ExchgParam^.T_SafetyCtrl.bStateTeachInToolCenter:=1;
		T_VisuQVis.ptrT_ExchgParam^.T_SafetyCtrl.bStateTeachInToolRight:=1;
		T_VisuQVis.ptrT_ExchgParam^.T_SafetyCtrl.bStateTeachInToolFeeder:=1;
		T_VisuQVis.ptrT_ExchgParam^.T_SafetyCtrl.bStateTeachInGrindFeeder:=1;
		T_VisuQVis.ptrT_ExchgParam^.T_StationCommon.iWireFeederRefIndexState:=1;
		IF T_Station.TControl.xActiveHardware THEN
			T_Station.TControl.xSecurityCircuitOn:=TRUE;
			T_Station.TControl.xSecurityCircuitOff:=FALSE;
		END_IF;
		T_Process.xEnable:=TRUE;
		QarxDigitalOutput[3]:=FALSE;	(* QxCtrlLampReleaseButton *)
	END_IF;

(****************************************************************************************************************************************************)
(***********                   start of the check for the hardware configuration changement and error during the startup                  ************)
(****************************************************************************************************************************************************)
(* Check changement of the Hardware Configuration *)
	IF T_StartUp.T_State.xCompleted AND NOT(xSwitchOffMachine) AND NOT(xSwitchOffMachineReady) THEN
		IF T_Station.TControl.xHardwareConfigError THEN
			xSwitchOffMachine:=TRUE;
		END_IF;
		IF xSwitchOffMachine THEN
			TONWaitSwitchOffMachine(IN:=FALSE);
			iStepSwitchOffMachine:=1;
		END_IF;
	END_IF;
	IF xSwitchOffMachine THEN
		TONWaitSwitchOffMachine(IN:=TRUE,PT:=T#5s);
		CASE iStepSwitchOffMachine OF
		1:	IF NOT(T_VisuQVis.T_CtrleVisu.xExecute) AND T_VisuQVis.T_CtrleVisu.xDone THEN
				T_NovRAM.T_Ctrle.xReset:=TRUE;
				T_VisuQVis.ptrT_ExchgParam^.T_TouchScreenBtPanel.iStateBtLeft:=0;
				T_VisuQVis.T_PlcParam.dwSetNewPage:=16#A;	(* Main Page wird aufgerufen *)
				T_VisuQVis.T_CtrleVisu.iFunction:=1;
				T_VisuQVis.T_CtrleVisu.xExecute:=TRUE;
				iStepSwitchOffMachine:=10;
			END_IF;
		10:	IF NOT(T_VisuQVis.T_CtrleVisu.xExecute) AND T_VisuQVis.T_CtrleVisu.xDone THEN
				T_StartUp.T_State.xBlockChangeMovementVisu:=TRUE;	(* Lock the navigation of the visu *)
				(* Overlay Message Error *)
				T_VisuQVis.ptrT_ExchgParam^.T_SafetyCtrl.bStateMessageError:=1;
				T_VisuQVis.ptrT_ExchgParam^.T_SafetyCtrl.bStateMessageInfo:=0;
				T_VisuQVis.ptrT_ExchgParam^.T_SafetyCtrl.bStateMessageWarning:=0;
				T_VisuQVis.ptrT_ExchgParam^.T_SafetyCtrl.iMsgErrorLine1:=19;	(* THE HARDWARE CONFIGURATION *)
				T_VisuQVis.ptrT_ExchgParam^.T_SafetyCtrl.iMsgErrorLine2:=19;	(* HAS BEEN CHANGED! *)
				T_VisuQVis.ptrT_ExchgParam^.T_SafetyCtrl.iMsgErrorLine3:=19;	(* THE MACHINE WILL BE SWITCHED OFF *)
				T_VisuQVis.ptrT_ExchgParam^.T_SafetyCtrl.iMsgErrorLine4:=19;	(* IN 5 SECONDS *)
				T_VisuQVis.ptrT_ExchgParam^.T_SafetyCtrl.xConfirmMsgError:=FALSE;
				T_VisuQVis.ptrT_ExchgParam^.T_SafetyCtrl.xBlockVisuObject:=TRUE;
				(* next step *)
				iStepSwitchOffMachine:=20;
			END_IF;
		20:	IF T_VisuQVis.ptrT_ExchgParam^.T_SafetyCtrl.xConfirmMsgError THEN
				T_VisuQVis.ptrT_ExchgParam^.T_SafetyCtrl.xBlockVisuObject:=FALSE;
				T_StartUp.T_State.xBlockChangeMovementVisu:=FALSE;	(* Unlock the navigation of the visu *)
				T_VisuQVis.ptrT_ExchgParam^.T_SafetyCtrl.bStateMessageError:=0;
				T_VisuQVis.ptrT_ExchgParam^.T_SafetyCtrl.xConfirmMsgError:=FALSE;
				iStepSwitchOffMachine:=1;
				xSwitchOffMachine:=FALSE;
				xSwitchOffMachineReady:=TRUE;
			END_IF;
		END_CASE;
		IF TONWaitSwitchOffMachine.Q  THEN
			T_VisuQVis.ptrT_ExchgParam^.T_SafetyCtrl.xBlockVisuObject:=FALSE;
			T_StartUp.T_State.xBlockChangeMovementVisu:=FALSE;	(* Unlock the navigation of the visu *)
			T_VisuQVis.ptrT_ExchgParam^.T_SafetyCtrl.bStateMessageError:=0;
			T_VisuQVis.ptrT_ExchgParam^.T_SafetyCtrl.xConfirmMsgError:=FALSE;
			iStepSwitchOffMachine:=1;
			xSwitchOffMachine:=FALSE;
			xSwitchOffMachineReady:=TRUE;
		END_IF;
	END_IF;
	IF xSwitchOffMachineReady THEN
		TONWaitSwitchOffMachine(IN:=FALSE);
		xSwitchOffMachineReady:=FALSE;
		xSwitchOffMachine:=FALSE;
		T_StartUp.T_State.xCompleted:=FALSE;
		xSetOutputDisable:=TRUE;
		T_VisuQVis.T_CtrleVisu.xReset:=TRUE;
		T_StartUp.T_Ctrle.xDone:=TRUE;
		T_StartUp.T_Ctrle.xErr:=FALSE;
		T_StartUp.T_Ctrle.udiErrorID:=0;
		xInitVisu:=FALSE;
		tTimeOutFunction:=T#0s;
		(* Start Booting *)
		T_StartUp.T_Ctrle.xExecute:=TRUE;
		T_StartUp.T_Ctrle.iFunction:=5;
	END_IF;

(* Check Hardware Error *)
	IF T_StartUp.T_State.xCompleted AND T_Station.TControl.xEnd AND NOT(T_Station.TControl.xError) AND T_Process.xEnd AND NOT(T_Process.xError) THEN
		xTmp:=	T_VisuQVis.T_CtrleAction.xDone AND
				(*T_VisuQVis.T_CtrleProcess.xDone AND
				T_VisuQVis.T_CtrleVisu.xDone AND*)
				(T_VisuQVis.ptrT_ExchgParam^.T_Visu.T_Message.iState <> 401);
		IF xTmp THEN
			diTmpErrorNr:=0;
			IF T_Station.THardware.TAxisToolLeft.T_CtrleSingle.xErr THEN
				diTmpErrorNr:=(T_Station.THardware.TAxisToolLeft.T_Config_Gen.iTyp * 1000000) + T_Station.THardware.TAxisToolLeft.T_CtrleSingle.udiErrorID;
			END_IF;
			IF T_Station.THardware.TAxisToolCenter.T_CtrleSingle.xErr AND xMicroRodActive THEN
				diTmpErrorNr:=(T_Station.THardware.TAxisToolCenter.T_Config_Gen.iTyp * 1000000) + T_Station.THardware.TAxisToolCenter.T_CtrleSingle.udiErrorID;
			END_IF;
			IF T_Station.THardware.TAxisToolRight.T_CtrleSingle.xErr THEN
				diTmpErrorNr:=(T_Station.THardware.TAxisToolRight.T_Config_Gen.iTyp * 1000000) + T_Station.THardware.TAxisToolRight.T_CtrleSingle.udiErrorID;
			END_IF;
			IF T_Station.THardware.TAxisToolFeeder.T_CtrleSingle.xErr THEN
				diTmpErrorNr:=(T_Station.THardware.TAxisToolFeeder.T_Config_Gen.iTyp * 1000000) + T_Station.THardware.TAxisToolFeeder.T_CtrleSingle.udiErrorID;
			END_IF;
			IF T_Station.THardware.TAxisGrindFeeder.T_CtrleSingle.xErr THEN
				diTmpErrorNr:=(T_Station.THardware.TAxisGrindFeeder.T_Config_Gen.iTyp * 1000000) + T_Station.THardware.TAxisGrindFeeder.T_CtrleSingle.udiErrorID;
			END_IF;
			IF (diTmpErrorNr <> 0) THEN
				FBErrorMessage(	diErrorNr:=diTmpErrorNr,
								T_ErrorList:=T_ErrorList);
				T_VisuQVis.ptrT_ExchgParam^.T_Visu.T_Message.sDynamicTextEnglish:=FBErrorMessage.sErrorTextEnglish;
				T_VisuQVis.ptrT_ExchgParam^.T_Visu.T_Message.sDynamicTextDeutsch:=FBErrorMessage.sErrorTextDeutsch;
				T_VisuQVis.ptrT_ExchgParam^.T_Visu.T_Message.sDynamicTextFrancais:=FBErrorMessage.sErrorTextFrancais;
				T_VisuQVis.ptrT_ExchgParam^.T_SafetyCtrl.diSetForceErrorNr:=diTmpErrorNr;
				T_VisuQVis.ptrT_ExchgParam^.T_SafetyCtrl.xSetForceError:=TRUE;
			END_IF;
		END_IF;
	END_IF;

(****************************************************************************************************************************************************)
(***********                                            end of the check for the hardware configuration changement                                               ************)
(****************************************************************************************************************************************************)

(* Manage BIOS Parameter *)
	IF T_StartUp.T_State.xPLCReady THEN
		FBBIOSPARAMETER(	dwBIOSPasswordPage:= 1,
							dwBIOSParameterPage:= 2,
							T_TwinSafeOut:= T_TwinSafeOut,
							T_Visu:= T_VisuQVis,
							T_HDD:= T_HDD,
							T_NovRam:= T_NovRam,
							T_CtrlePanel:= T_CtrlePanel,
							T_DeviceID:= T_DeviceID,
							T_BoxID:= T_BoxID,
							T_Profile:= T_Profile);
	END_IF;

(****************************************************************************************************************************************************)
(***********                                                      start of the execution for the function of the start up                                                          ************)
(****************************************************************************************************************************************************)
(* Function Init PLC *)
	IF xInitVisu AND NOT(xEmergency) AND NOT(xNoAirPressure) AND NOT(xNodeFailCANOpen) THEN
		CASE iStepFunction OF
		1:	T_VisuQVis.T_CtrleVisu.xActive:=TRUE;
			T_VisuQVis.T_CtrleVisu.xReset:=TRUE;
			(* next step *)
			iStepFunction:=10;
		(* Confirm Reset *)
		10:	IF T_VisuQVis.T_CtrleVisu.xDone THEN
				T_StartUp.T_State.xPLCReady:=TRUE;
				(* next step *)
				iStepFunction:=90;
			END_IF
		(* end function or time out *)
		90:	T_StartUp.T_Ctrle.xDone:=TRUE;
			T_StartUp.T_Ctrle.xErr:=FALSE;
			T_StartUp.T_Ctrle.udiErrorID:=0;
			xInitVisu:=FALSE;
			tTimeOutFunction:=T#0s;
			(* Start Read Hardware *)
			T_StartUp.T_Ctrle.xExecute:=TRUE;
			T_StartUp.T_Ctrle.iFunction:=8;
		END_CASE
	END_IF

(* Function ReadHardware with NovRAM Parameter *)
	IF xReadHardware AND NOT(xEmergency) AND NOT(xNoAirPressure) AND NOT(xNodeFailCANOpen) THEN
		CASE iStepFunction OF
		(* Start station, reset FB *)
		1:	T_HDD.T_Ctrle.xReset:=TRUE;
			T_DeviceID.T_Ctrle.xReset:=TRUE;
			T_BoxID.T_Ctrle.xReset:=TRUE;
			T_NovRAM.T_Ctrle.xReset:=TRUE;
			T_Profile.T_Ctrle.xReset:=TRUE;
			(* next step *)
			iStepFunction:=10;
		(* waiting reset confirmation *)
		10:	xTmp:=	T_HDD.T_Ctrle.xDone
					AND T_DeviceID.T_Ctrle.xDone
					AND T_NovRAM.T_Ctrle.xDone
					AND T_BoxID.T_Ctrle.xDone;
			IF xTmp THEN  iStepFunction:=20; END_IF
		(* Init. device name *)
		20:	(* PLC name *)
			T_DeviceID.T_CX1020.sDeviceName:='CX1000_PLC';
			(* feldbus name *)
			T_DeviceID.T_CANOpenMaster.sDeviceName:='CANOpenMaster';
			T_DeviceID.T_CANOpenMaster.xDeviceOption:=TRUE;
			T_DeviceID.T_LightbusMaster.sDeviceName:='LightbusMaster';
			T_DeviceID.T_LightbusMaster.xDeviceOption:=TRUE;
			(* NovRAM *)
			T_DeviceID.T_NovRAM.sDeviceName:='NovRAM';
			(* read device ID *)
			T_DeviceID.T_Ctrle.xExecute:=TRUE;
			(* next step *)
			iStepFunction:=30;
		(* waiting ID confirmation, Start BoxID *)
		30:	IF NOT(T_DeviceID.T_Ctrle.xExecute) AND T_DeviceID.T_Ctrle.xDone THEN iStepFunction:=40; END_IF
		(* waiting Box ID confirmation *)
		40:	IF NOT(T_BoxID.T_Ctrle.xExecute) AND T_BoxID.T_Ctrle.xDone THEN
				(* next step *)
				iStepFunction:=50;
			END_IF
		50:	T_NovRAM.T_Ctrle.iFunction:=1;
			T_NovRam.T_Ctrle.xBlockReadFirstTime:=FALSE;
			T_NovRAM.T_Ctrle.xExecute:=TRUE;
			iStepFunction:=60;
		60:	IF NOT(T_NovRAM.T_Ctrle.xExecute) AND T_NovRAM.T_Ctrle.xDone THEN
				T_VisuQVis.ptrT_ExchgParam^.T_StationCommon.iConfigAxisType:=T_NovRAM.T_Data.T_Standard.T_MachineConfig.iConfigAxisType;
				T_VisuQVis.ptrT_ExchgParam^.T_StationCommon.iConfigMachineType:=T_NovRAM.T_Data.T_Standard.T_MachineConfig.iConfigMachineType;
				T_VisuQVis.ptrT_ExchgParam^.T_StationCommon.iConfigVisuNavigation:=T_NovRAM.T_Data.T_Standard.T_MachineConfig.iConfigVisuNavigation;
				T_VisuQVis.ptrT_ExchgParam^.T_StationCommon.rConfigMaxToolLength:=T_NovRAM.T_Data.T_Standard.T_MachineConfig.rConfigMaxToolLength;
				(*08.12.2010 KFS:	{	*)
				T_VisuQVis.ptrT_ExchgParam^.T_StationCommon.rConfigMaxToolLengthOriginal:=T_NovRAM.T_Data.T_Standard.T_MachineConfig.rConfigMaxToolLengthOriginal;
				(*08.12.2010 KFS:	}	*)
				T_VisuQVis.T_CtrleVisu.xReset:=TRUE;
				iStepFunction:=70;
			END_IF;
		(* end function or time out *)
		70:	IF T_VisuQVis.T_CtrleVisu.xDone THEN
				T_VisuQVis.ptrT_ExchgParam^.T_Config.xNoTouchScreenBtPanel:=TRUE;
				T_StartUp.T_Ctrle.xDone:=TRUE;
				T_StartUp.T_Ctrle.xErr:=FALSE;
				T_StartUp.T_Ctrle.udiErrorID:=0;
				xReadHardware:=FALSE;
				tTimeOutFunction:=T#0s;
				(* Start Boot *)
				T_StartUp.T_Ctrle.xExecute:=TRUE;
				T_StartUp.T_Ctrle.iFunction:=5;
			END_IF;
		END_CASE;
	END_IF;

(* Function Start Booting *)
	IF xStartBooting AND NOT(xEmergency) AND NOT(xNoAirPressure) AND NOT(xNodeFailCANOpen) THEN
		T_VisuQVis.ptrT_ExchgParam^.T_Visu.iLoadingStartPage:=1;
		CASE iStepFunction OF
		1:	IF (T_NovRam.T_Data.T_Standard.T_MachineConfig.iConfigMachineType = 2) THEN
				xMicroRodActive:=TRUE;
			ELSE
				xMicroRodActive:=FALSE;
			END_IF;
			T_TwinSafeCtrleOUT.xTwinSAFE_Run:=FALSE;	(* Stop TwinSafe Groupe *)
			QarxDigitalOutput[1]:=FALSE;	(* QxCtrlLampStartButton *)
			QarxDigitalOutput[2]:=FALSE;	(* QxCtrlLampStopButton *)
			QarxDigitalOutput[3]:=FALSE;	(* QxCtrlLampReleaseButton *)
			IF NOT(T_TwinSafeIn.IxEmergencyStopMachine) OR NOT(T_TwinSafeIn.IxEmergencyStopStuder) THEN		(* check state of emergency button *)
				(* Overlay Message Error *)
				T_VisuQVis.ptrT_ExchgParam^.T_SafetyCtrl.bStateMessageError:=1;
				T_VisuQVis.ptrT_ExchgParam^.T_SafetyCtrl.bStateMessageInfo:=0;
				T_VisuQVis.ptrT_ExchgParam^.T_SafetyCtrl.bStateMessageWarning:=0;
				T_VisuQVis.ptrT_ExchgParam^.T_SafetyCtrl.iMsgErrorLine1:=1;	(* EMERGENCY STOP BUTTON IS ACITVE! *)
				T_VisuQVis.ptrT_ExchgParam^.T_SafetyCtrl.iMsgErrorLine2:=1;	(* PLEASE RELEASE THIS BUTTON *)
				T_VisuQVis.ptrT_ExchgParam^.T_SafetyCtrl.iMsgErrorLine3:=1;	(* AND AFTER CONFIRM THIS MESSAGE *)
				T_VisuQVis.ptrT_ExchgParam^.T_SafetyCtrl.iMsgErrorLine4:=1;	(*  *)
				T_VisuQVis.ptrT_ExchgParam^.T_SafetyCtrl.xConfirmMsgError:=FALSE;
				T_VisuQVis.ptrT_ExchgParam^.T_SafetyCtrl.xBlockVisuObject:=TRUE;
				(* next step *)
				iStepFunction:=10;
			ELSE
				(* next step *)
				iStepFunction:=11;
				TONWaitResetOutput(IN:=FALSE);
			END_IF;
			T_VisuQVis.ptrT_ExchgParam^.T_Visu.T_Level.iPwSystem:=999;	(* Releas System Level *)
			T_VisuQVis.ptrT_ExchgParam^.T_Visu.T_Level.iActLevel:=1;
		10:	IF T_VisuQVis.ptrT_ExchgParam^.T_SafetyCtrl.xConfirmMsgError THEN
				T_VisuQVis.ptrT_ExchgParam^.T_SafetyCtrl.xBlockVisuObject:=FALSE;
				T_VisuQVis.ptrT_ExchgParam^.T_SafetyCtrl.bStateMessageError:=0;
				T_VisuQVis.ptrT_ExchgParam^.T_SafetyCtrl.xConfirmMsgError:=FALSE;
				(* next step *)
				iStepFunction:=1;
			END_IF;
		11:	TONWaitResetOutput(IN:=TRUE,PT:=T#500ms);
			IF TONWaitResetOutput.Q THEN
				TONWaitResetOutput(IN:=FALSE);
				iStepFunction:=20;
			END_IF;
		20:	xStartCheck:=FALSE;
			T_TwinSafeCtrleOUT.xTwinSAFE_Run:=TRUE;	(* Start TwinSafe Groupe *)
			TONWaitResetOutput(IN:=FALSE);
			(* next step *)
			iStepFunction:=21;
		21:	TONWaitResetOutput(IN:=TRUE,PT:=T#200ms);
			IF TONWaitResetOutput.Q THEN
				IF T_TwinSafeCtrleIN.xTwinSAFE_Group_FB_Error OR T_TwinSafeCtrleIN.xTwinSAFE_Group_COM_Error THEN
					T_TwinSafeCtrleOUT.xTwinSAFE_Reset:=TRUE;
					TONWaitResetOutput(IN:=FALSE);
					iStepFunction:=22;
					RETURN;
				END_IF;
				TONWaitResetOutput(IN:=FALSE);
				iStepFunction:=24;
			END_IF;
		22:	TONWaitResetOutput(IN:=TRUE,PT:=T#200ms);
			IF TONWaitResetOutput.Q THEN
				T_TwinSafeCtrleOUT.xTwinSAFE_Reset:=FALSE;
				T_TwinSafeCtrleOUT.xTwinSAFE_Run:=FALSE;	(* Stop TwinSafe Groupe *)
				TONWaitResetOutput(IN:=FALSE);
				iStepFunction:=23;
			END_IF;
		23:	TONWaitResetOutput(IN:=TRUE,PT:=T#200ms);
			IF TONWaitResetOutput.Q THEN
				TONWaitResetOutput(IN:=FALSE);
				iStepFunction:=20;
			END_IF;
		24:	IF T_TwinSafeIn.IxReadyToolLeft OR T_TwinSafeIn.IxReadyToolCenter OR T_TwinSafeIn.IxReadyToolRight OR T_TwinSafeIn.IxReadyToolFeeder OR T_TwinSafeIn.IxReadyGrindFeeder THEN
				T_Station.TControl.xResetHardware:=TRUE;
				iStepFunction:=25;
			ELSE
				iStepFunction:=30;
			END_IF;
		25:	IF NOT(T_Station.TControl.xResetHardware) THEN
				iStepFunction:=30;
			END_IF;
		30:	QarxDigitalOutput[3]:=TRUE;	(* QxCtrlLampReleaseButton *)
			T_VisuQVis.ptrT_ExchgParam^.T_SafetyCtrl.iStateStartPage:=1;	(* Press external Quit Button *)
			(* next step *)
			iStepFunction:=40;
		40:	T_VisuQVis.ptrT_ExchgParam^.T_SafetyCtrl.iStateStartPage:=1;	(* Press external Quit Button *)
			IF NOT(T_TwinSafeIn.IxPowerSupplyEcoStep) THEN
				QarxDigitalOutput[4]:=TRUE;	(* QxCtrlLampCurEcoButton *)
				T_VisuQVis.ptrT_ExchgParam^.T_SafetyCtrl.iStateStartPage:=4;	(* Message: Release AxesCurrentButton *)
				RETURN;	(* Do nothing if the Button AxesCurrent is Active *)
			END_IF;
			IF RisingEdgeQuitButton.Q THEN		(* Wait until the Operator press the external quit button *)
				QarxDigitalOutput[3]:=FALSE;	(* QxCtrlLampReleaseButton *)
				T_VisuQVis.ptrT_ExchgParam^.T_SafetyCtrl.iStateStartPage:=0;	(* No Text *)
				xDeleteErrorMessage:=TRUE;	(* Reset the line message error *)
				TONWaitCircuitOn(IN:=FALSE);
				(* next step *)
				iStepFunction:=50;
			END_IF;
		50:	TONWaitCircuitOn(IN:=TRUE,PT:=T#500ms);
			IF TONWaitCircuitOn.Q THEN
				TONWaitCircuitOn(IN:=FALSE);
				(* next step *)
				iStepFunction:=60;
			END_IF;
		60:	IF NOT(T_TwinSafeIn.IxPowerSupplyEcoStep) THEN	(* Check if the power supply of the EcoStep is switched Off *)
				T_TwinSafeCtrleOUT.xTwinSAFE_Run:=FALSE;	(* Stop TwinSafe Groupe *)
				(* Overlay Message Error *)
				T_VisuQVis.ptrT_ExchgParam^.T_SafetyCtrl.bStateMessageError:=1;
				T_VisuQVis.ptrT_ExchgParam^.T_SafetyCtrl.bStateMessageInfo:=0;
				T_VisuQVis.ptrT_ExchgParam^.T_SafetyCtrl.bStateMessageWarning:=0;
				T_VisuQVis.ptrT_ExchgParam^.T_SafetyCtrl.iMsgErrorLine1:=4;	(* FOR BOOTING THE MACHINE *)
				T_VisuQVis.ptrT_ExchgParam^.T_SafetyCtrl.iMsgErrorLine2:=4;	(* SWITCH ON THE POWER SUPPLY ECOSTEP *)
				T_VisuQVis.ptrT_ExchgParam^.T_SafetyCtrl.iMsgErrorLine3:=4;	(* CONFIRM THIS MESSAGE AND  *)
				T_VisuQVis.ptrT_ExchgParam^.T_SafetyCtrl.iMsgErrorLine4:=4;	(* PRESS THE  RELEASE BUTTON *)
				T_VisuQVis.ptrT_ExchgParam^.T_SafetyCtrl.xConfirmMsgError:=FALSE;
				T_VisuQVis.ptrT_ExchgParam^.T_SafetyCtrl.xBlockVisuObject:=TRUE;
				(* next step *)
				iStepFunction:=70;
			ELSE
				IF NOT(T_TwinSafeOut.QxContactor_K3) AND NOT(T_TwinSafeOut.QxContactor_K4) THEN
					T_TwinSafeCtrleOUT.xTwinSAFE_Run:=FALSE;	(* Stop TwinSafe Groupe *)
					T_VisuQVis.ptrT_ExchgParam^.T_SafetyCtrl.bStateMessageError:=1;
					T_VisuQVis.ptrT_ExchgParam^.T_SafetyCtrl.bStateMessageInfo:=0;
					T_VisuQVis.ptrT_ExchgParam^.T_SafetyCtrl.bStateMessageWarning:=0;
					T_VisuQVis.ptrT_ExchgParam^.T_SafetyCtrl.xConfirmMsgError:=FALSE;
					T_VisuQVis.ptrT_ExchgParam^.T_SafetyCtrl.xBlockVisuObject:=TRUE;
					IF NOT(T_TwinSafeIn.IxReadyToolLeft) AND ((NOT(T_TwinSafeIn.IxReadyToolCenter) AND xMicroRodActive) OR NOT(xMicroRodActive)) AND
					     NOT(T_TwinSafeIn.IxReadyToolRight) AND NOT(T_TwinSafeIn.IxReadyToolFeeder) AND NOT(T_TwinSafeIn.IxReadyGrindFeeder) THEN
						(* Overlay Message Error *)
						T_VisuQVis.ptrT_ExchgParam^.T_SafetyCtrl.iMsgErrorLine1:=6;	(* THE CONNECTOR K3 OR K4 *)
						T_VisuQVis.ptrT_ExchgParam^.T_SafetyCtrl.iMsgErrorLine2:=6;	(* ARE NOT WORKING PROPERLY *)
						T_VisuQVis.ptrT_ExchgParam^.T_SafetyCtrl.iMsgErrorLine3:=6;	(* PLEASE CONFIRM AND TRY AGAIN  *)
						T_VisuQVis.ptrT_ExchgParam^.T_SafetyCtrl.iMsgErrorLine4:=6;	(*OTHERWISE CHECK THE EQUIPMENT *)
					ELSE
						T_VisuQVis.ptrT_ExchgParam^.T_SafetyCtrl.iMsgErrorLine1:=21;	(* AT LEAST ONE CANOPEN CONTROLLER FAILED! *)
						T_VisuQVis.ptrT_ExchgParam^.T_SafetyCtrl.iMsgErrorLine2:=21;	(* PLEASE CHECK THE ECOSTEP AXIS *)
						T_VisuQVis.ptrT_ExchgParam^.T_SafetyCtrl.iMsgErrorLine3:=21;	(* AND CONFIRM THIS MESSAGE *)
						T_VisuQVis.ptrT_ExchgParam^.T_SafetyCtrl.iMsgErrorLine4:=21;	(*  *)
						FBErrorMessage(	diErrorNr:=6,		(* At least one Ecostep CANOpen Controller failed! *)
										T_ErrorList:=T_ErrorList);
						T_VisuQVis.ptrT_ExchgParam^.T_Visu.T_Message.sDynamicTextEnglish:=FBErrorMessage.sErrorTextEnglish;
						T_VisuQVis.ptrT_ExchgParam^.T_Visu.T_Message.sDynamicTextDeutsch:=FBErrorMessage.sErrorTextDeutsch;
						T_VisuQVis.ptrT_ExchgParam^.T_Visu.T_Message.sDynamicTextFrancais:=FBErrorMessage.sErrorTextFrancais;
						(* Safe the error *)
						T_VisuQVis.ptrT_ExchgParam^.T_SafetyCtrl.diSetForceErrorNr:=6;
						T_VisuQVis.ptrT_ExchgParam^.T_SafetyCtrl.xSetForceError:=TRUE;
					END_IF;
					(* next step *)
					iStepFunction:=70;
				ELSE
					TONWaitCircuitOn(IN:=FALSE);
					(* next step *)
					iStepFunction:=80;
				END_IF;
			END_IF;
		70:	IF T_VisuQVis.ptrT_ExchgParam^.T_SafetyCtrl.xConfirmMsgError THEN
				T_VisuQVis.ptrT_ExchgParam^.T_SafetyCtrl.xBlockVisuObject:=FALSE;
				T_VisuQVis.ptrT_ExchgParam^.T_SafetyCtrl.bStateMessageError:=0;
				T_VisuQVis.ptrT_ExchgParam^.T_SafetyCtrl.xConfirmMsgError:=FALSE;
				xCheckSecurityDoor:=FALSE;
				TONWaitCircuitOn(IN:=FALSE);
				(* next step *)
				iStepFunction:=1;
			END_IF;
		80:	TONWaitCircuitOn(IN:=TRUE,PT:=T#2000ms);
			IF TONWaitCircuitOn.Q OR IarxDigitalInput[4] THEN	(* Check if the pressure of the air is present *)
				TONWaitCircuitOn(IN:=FALSE);
				(* next step *)
				iStepFunction:=90;
			END_IF;
			xCheckSecurityDoor:=TRUE;
		90:	IF NOT(IarxDigitalInput[4]) THEN		(* check state of air pressure *)
				xCheckSecurityDoor:=FALSE;
				T_TwinSafeCtrleOUT.xTwinSAFE_Run:=FALSE;	(* Stop TwinSafe Groupe *)
				(* Overlay Message Error *)
				T_VisuQVis.ptrT_ExchgParam^.T_SafetyCtrl.bStateMessageError:=1;
				T_VisuQVis.ptrT_ExchgParam^.T_SafetyCtrl.bStateMessageInfo:=0;
				T_VisuQVis.ptrT_ExchgParam^.T_SafetyCtrl.bStateMessageWarning:=0;
				T_VisuQVis.ptrT_ExchgParam^.T_SafetyCtrl.iMsgErrorLine1:=2;	(* NO AIR PRESSURE! *)
				T_VisuQVis.ptrT_ExchgParam^.T_SafetyCtrl.iMsgErrorLine2:=2;	(* PLEASE ACTIVATE THE AIR PRESSURE *)
				T_VisuQVis.ptrT_ExchgParam^.T_SafetyCtrl.iMsgErrorLine3:=2;	(* AND AFTER CONFIRM THIS MESSAGE *)
				T_VisuQVis.ptrT_ExchgParam^.T_SafetyCtrl.iMsgErrorLine4:=2;	(*  *)
				T_VisuQVis.ptrT_ExchgParam^.T_SafetyCtrl.xConfirmMsgError:=FALSE;
				T_VisuQVis.ptrT_ExchgParam^.T_SafetyCtrl.xBlockVisuObject:=TRUE;
				FBErrorMessage(	diErrorNr:=7,		(* No Air Pressure *)
							T_ErrorList:=T_ErrorList);
				T_VisuQVis.ptrT_ExchgParam^.T_Visu.T_Message.sDynamicTextEnglish:=FBErrorMessage.sErrorTextEnglish;
				T_VisuQVis.ptrT_ExchgParam^.T_Visu.T_Message.sDynamicTextDeutsch:=FBErrorMessage.sErrorTextDeutsch;
				T_VisuQVis.ptrT_ExchgParam^.T_Visu.T_Message.sDynamicTextFrancais:=FBErrorMessage.sErrorTextFrancais;
				(* Safe the error *)
				T_VisuQVis.ptrT_ExchgParam^.T_SafetyCtrl.diSetForceErrorNr:=7;
				T_VisuQVis.ptrT_ExchgParam^.T_SafetyCtrl.xSetForceError:=TRUE;
				(* next step *)
				iStepFunction:=100;
			ELSE
				(* next step *)
				iStepFunction:=110;
			END_IF;
		100:	IF T_VisuQVis.ptrT_ExchgParam^.T_SafetyCtrl.xConfirmMsgError THEN
				T_VisuQVis.ptrT_ExchgParam^.T_SafetyCtrl.xBlockVisuObject:=FALSE;
				T_VisuQVis.ptrT_ExchgParam^.T_SafetyCtrl.bStateMessageError:=0;
				T_VisuQVis.ptrT_ExchgParam^.T_SafetyCtrl.xConfirmMsgError:=FALSE;
				(* next step *)
				iStepFunction:=20;
			END_IF;
		110:	QarxDigitalOutput[1]:=TRUE;	(* QxCtrlLampStartButton *)
			T_VisuQVis.ptrT_ExchgParam^.T_SafetyCtrl.iStateStartPage:=2;	(* Press external start button *)
			(* next step *)
			iStepFunction:=120;
		120:	QarxDigitalOutput[1]:=TRUE;	(* QxCtrlLampStartButton *)
			T_VisuQVis.ptrT_ExchgParam^.T_SafetyCtrl.iStateStartPage:=2;	(* Press external start button *)
			IF RisingEdgeStartButton.Q THEN		(* Wait until the Operator press the external start button *)
				QarxDigitalOutput[1]:=FALSE;	(* QxCtrlLampStartButton *)
				T_VisuQVis.ptrT_ExchgParam^.T_SafetyCtrl.iStateStartPage:=0;
				xDeleteErrorMessage:=TRUE;	(* Reset the line message error *)
				(* next step *)
				iStepFunction:=130;
			END_IF;
			IF NOT(T_TwinSafeIn.IxPowerSupplyEcoStep) THEN	(* Check if the power supply of the EcoStep is switched Off *)
				(* next step *)
				iStepFunction:=60;
				RETURN;
			END_IF;
		130:	IF IarxDigitalInput[3] THEN	(* Check if the key switch is active *)
				(* Overlay Message Error *)
				T_VisuQVis.ptrT_ExchgParam^.T_SafetyCtrl.bStateMessageError:=1;
				T_VisuQVis.ptrT_ExchgParam^.T_SafetyCtrl.bStateMessageInfo:=0;
				T_VisuQVis.ptrT_ExchgParam^.T_SafetyCtrl.bStateMessageWarning:=0;
				T_VisuQVis.ptrT_ExchgParam^.T_SafetyCtrl.iMsgErrorLine1:=5;	(* FOR BOOTING THE MACHINE IT IS MANDATORY *)
				T_VisuQVis.ptrT_ExchgParam^.T_SafetyCtrl.iMsgErrorLine2:=5;	(* THAT YOU SWITCH OFF THE KEY SWITCH *)
				T_VisuQVis.ptrT_ExchgParam^.T_SafetyCtrl.iMsgErrorLine3:=5;	(* CONFIRM THIS MESSAGE AND TRY AGAIN *)
				T_VisuQVis.ptrT_ExchgParam^.T_SafetyCtrl.iMsgErrorLine4:=5;	(* TO PRESS THE EXTERNAL START BUTTON *)
				T_VisuQVis.ptrT_ExchgParam^.T_SafetyCtrl.xConfirmMsgError:=FALSE;
				T_VisuQVis.ptrT_ExchgParam^.T_SafetyCtrl.xBlockVisuObject:=TRUE;
				(* next step *)
				iStepFunction:=140;
			ELSE
				(* next step *)
				iStepFunction:=150;
			END_IF;
		140:	IF T_VisuQVis.ptrT_ExchgParam^.T_SafetyCtrl.xConfirmMsgError THEN
				T_VisuQVis.ptrT_ExchgParam^.T_SafetyCtrl.xBlockVisuObject:=FALSE;
				T_VisuQVis.ptrT_ExchgParam^.T_SafetyCtrl.bStateMessageError:=0;
				T_VisuQVis.ptrT_ExchgParam^.T_SafetyCtrl.xConfirmMsgError:=FALSE;
				(* next step *)
				iStepFunction:=110;
			END_IF;
			IF (NOT(T_TwinSafeOut.QxContactor_K3) OR NOT(T_TwinSafeOut.QxContactor_K4)) THEN
				T_VisuQVis.ptrT_ExchgParam^.T_SafetyCtrl.xBlockVisuObject:=FALSE;
				T_VisuQVis.ptrT_ExchgParam^.T_SafetyCtrl.bStateMessageError:=0;
				T_VisuQVis.ptrT_ExchgParam^.T_SafetyCtrl.xConfirmMsgError:=FALSE;
				(* next step *)
				iStepFunction:=1;
			END_IF;
		150:	(* Start Booting is ended, the machine has now the right state to boot the machine *)
			IF NOT(T_TwinSafeIn.IxPowerSupplyEcoStep) THEN	(* Check if the power supply of the EcoStep is switched Off *)
				(* next step *)
				iStepFunction:=60;
				RETURN;
			END_IF;
			xCheckSecurityDoor:=FALSE;
			xStartBooting:=FALSE;
			(* Start Loading *)
			T_StartUp.T_Ctrle.xExecute:=TRUE;
			T_StartUp.T_Ctrle.iFunction:=2;
		END_CASE;
	END_IF;

(* Function start loading *)
	IF xLoading AND NOT(xEmergency) AND NOT(xNoAirPressure) AND NOT(xNodeFailCANOpen) THEN
		(* Timer bargraph *)
		IF (iStepFunction < 999) THEN
			T_VisuQVis.ptrT_ExchgParam^.T_SafetyCtrl.iStateStartPage:=3;	(* Machine is booting *)
			TONStartUp(IN:=TRUE,PT:=tTimeStartUp);
			IF TONStartUp.Q THEN
				TONStartUp(IN:=FALSE);
				IF (T_VisuQVis.ptrT_ExchgParam^.T_Visu.iLoadingStartPage <=100) THEN
					T_VisuQVis.ptrT_ExchgParam^.T_Visu.iLoadingStartPage:=T_VisuQVis.ptrT_ExchgParam^.T_Visu.iLoadingStartPage +1; END_IF
			END_IF;
		END_IF;
		IF NOT(T_TwinSafeIn.IxPowerSupplyEcoStep) AND (T_VisuQVis.T_PlcParam.dwActualPage = 0) THEN	(* Check if the power supply of the EcoStep is switched Off *)
			T_Station.TControl.xEnable:=FALSE;
			xLoading:=FALSE;
			xStartBooting:=TRUE;
			tTimeOutFunction:=T#0s;	(* deactivate the time out *)
			(* next step *)
			iStepFunction:=60;
			RETURN;
		END_IF;
		CASE iStepFunction OF
		(* Check *)
		1:	 IF T_StartUp.T_State.xPLCReady THEN iStepFunction:=10; END_IF
		(* Init. Visu and Set Power *)
		10:	xDeleteErrorMessage:=TRUE;	(* Reset the line message error *)
			T_VisuQVis.T_PlcParam.dwSetNewPage:=16#0;
			T_VisuQVis.T_CtrleVisu.xReset:=TRUE;
			T_VisuQVis.T_CtrleVisu.xExecute:=TRUE;
			T_VisuQVis.T_CtrleVisu.iFunction:=1;
			(* Init. timer *)
			TimerDelayStartStation(IN:=FALSE);
			(* next Step *)
			iStepFunction:=20;
		(* Delay before start station *)
		20:	TimerDelayStartStation(IN:=TRUE, PT:=T#200ms);
			IF TimerDelayStartStation.Q THEN
				(* Init. timer *)
				TimerDelayStartStation(IN:=FALSE);
				(* Next step *)
				iStepFunction:=30;
			END_IF;
		30:	(* Check NodeState of the CANOpen for the Ecostep Axis *)
			xTmp:=	(T_AxisNodeState.bToolLeftNodeState <> 0) OR
					((T_AxisNodeState.bToolCenterNodeState <> 0) AND xMicroRodActive) OR
					(T_AxisNodeState.bToolRightNodeState <> 0) OR
					(T_AxisNodeState.bToolFeederNodeState <> 0) OR
					(T_AxisNodeState.bGrindFeederNodeState <> 0);
			IF xTmp THEN
				(* next step *)
				iStepFunction:=40;	(* At least one CANOpen Controller from the Ecostep Axis failed *)
			ELSE
				(* next step *)
				iStepFunction:=100;
			END_IF;
		(* Error CanOpen-->Ventilinsel *)
		40:	FBErrorMessage(	diErrorNr:=6,		(* At least one Ecostep CANOpen Controller failed! *)
							T_ErrorList:=T_ErrorList);
			T_VisuQVis.ptrT_ExchgParam^.T_Visu.T_Message.sDynamicTextEnglish:=FBErrorMessage.sErrorTextEnglish;
			T_VisuQVis.ptrT_ExchgParam^.T_Visu.T_Message.sDynamicTextDeutsch:=FBErrorMessage.sErrorTextDeutsch;
			T_VisuQVis.ptrT_ExchgParam^.T_Visu.T_Message.sDynamicTextFrancais:=FBErrorMessage.sErrorTextFrancais;
			(* Safe the error *)
			T_VisuQVis.ptrT_ExchgParam^.T_SafetyCtrl.diSetForceErrorNr:=6;
			T_VisuQVis.ptrT_ExchgParam^.T_SafetyCtrl.xSetForceError:=TRUE;
			iStepFunction:=999;
		100:	T_Station.TControl.xActiveStation:=TRUE;
			iStepFunction:=200;
		200:	T_Station.TControl.xEnable:=TRUE;
			iStepFunction:=300;
		300:	IF T_Station.TControl.xEnd AND T_Station.TControl.xError THEN
				FBErrorMessage(	diErrorNr:=T_Station.TControl.diErrorNr,
								T_ErrorList:=T_ErrorList);
				T_VisuQVis.ptrT_ExchgParam^.T_Visu.T_Message.sDynamicTextEnglish:=FBErrorMessage.sErrorTextEnglish;
				T_VisuQVis.ptrT_ExchgParam^.T_Visu.T_Message.sDynamicTextDeutsch:=FBErrorMessage.sErrorTextDeutsch;
				T_VisuQVis.ptrT_ExchgParam^.T_Visu.T_Message.sDynamicTextFrancais:=FBErrorMessage.sErrorTextFrancais;
				(* Safe the error *)
				T_VisuQVis.ptrT_ExchgParam^.T_SafetyCtrl.diSetForceErrorNr:=T_Station.TControl.diErrorNr;
				T_VisuQVis.ptrT_ExchgParam^.T_SafetyCtrl.xSetForceError:=TRUE;
				iStepFunction:=999;
				RETURN;
			END_IF;
			IF T_Station.TControl.xEnd AND T_Station.TControl.xRdy THEN
				T_VisuQVis.ptrT_ExchgParam^.T_StationCommon.T_ToolLeftSoftwareInfo:=T_Station.THardware.TAxisToolLeft.T_SoftwareDetails;
				T_VisuQVis.ptrT_ExchgParam^.T_StationCommon.T_ToolCenterSoftwareInfo:=T_Station.THardware.TAxisToolCenter.T_SoftwareDetails;
				T_VisuQVis.ptrT_ExchgParam^.T_StationCommon.T_ToolRightSoftwareInfo:=T_Station.THardware.TAxisToolRight.T_SoftwareDetails;
				T_VisuQVis.ptrT_ExchgParam^.T_StationCommon.T_ToolFeederSoftwareInfo:=T_Station.THardware.TAxisToolFeeder.T_SoftwareDetails;
				T_VisuQVis.ptrT_ExchgParam^.T_StationCommon.T_GrindFeederSoftwareInfo:=T_Station.THardware.TAxisGrindFeeder.T_SoftwareDetails;
				iStepFunction:=310;
			END_IF;
		310:	T_Process.xEnable:=TRUE;
			iStepFunction:=320;
		320:	IF T_Process.xRdy AND T_Process.xEnd THEN
				iStepFunction:=330;
			END_IF;
		330:	T_VisuQVis.ptrT_ExchgParam^.T_StationCommon.T_InfoProcess.iProfile:=T_NovRam.T_Data.T_Standard.T_InfoProcess.iProfile;
			T_VisuQVis.ptrT_ExchgParam^.T_StationCommon.T_InfoProcess.sProfileName:=T_NovRam.T_Data.T_Standard.T_InfoProcess.sProfileName;
			T_VisuQVis.ptrT_ExchgParam^.T_ProfileCommon.T_Id.iNumber:=T_NovRam.T_Data.T_Standard.T_InfoProcess.iProfile;
			T_VisuQVis.ptrT_ExchgParam^.T_ProfileCommon.T_Id.sName:=T_NovRam.T_Data.T_Standard.T_InfoProcess.sProfileName;
			T_VisuQVis.T_CtrleAction.xExecute:=TRUE;
			T_VisuQVis.T_CtrleAction.iFunction:=1001;
			iStepFunction:=340;
		340:	IF NOT(T_VisuQVis.T_CtrleAction.xExecute) AND T_VisuQVis.T_CtrleAction.xDone THEN
				T_VisuQVis.T_CtrleAction.xResetParaListValue:=TRUE;
				iStepFunction:=400;
			END_IF;
		400:	IF NOT(T_VisuQVis.T_CtrleAction.xResetParaListValue) THEN
				IF T_VisuQVis.T_CtrleAction.xDone THEN iStepFunction:=984; END_IF;
				IF T_VisuQVis.T_CtrleAction.xErr THEN iStepFunction:=999; END_IF
				IF T_VisuQVis.T_CtrleAction.xDone OR T_VisuQVis.T_CtrleAction.xErr THEN
					T_VisuQVis.T_PlcParam.dwSetNewPage:=16#A;	(* Main Page wird aufgerufen *)
					T_VisuQVis.T_CtrleVisu.iFunction:=1;
					T_VisuQVis.T_CtrleVisu.xExecute:=TRUE;
				END_IF;
			END_IF;
		984:	tTimeOutFunction:=T#0s;	(* deactivate the time out *)
			(* Overlay Message Error *)
			T_VisuQVis.ptrT_ExchgParam^.T_SafetyCtrl.bStateMessageError:=0;
			T_VisuQVis.ptrT_ExchgParam^.T_SafetyCtrl.bStateMessageInfo:=1;
			T_VisuQVis.ptrT_ExchgParam^.T_SafetyCtrl.bStateMessageWarning:=0;
			T_VisuQVis.ptrT_ExchgParam^.T_SafetyCtrl.iMsgInfoLine1:=1;	(* BOOTING OF THE MACHINE COMPLEATED! *)
			T_VisuQVis.ptrT_ExchgParam^.T_SafetyCtrl.iMsgInfoLine2:=1;	(* CONFIRM AND THE MACHINE *)
			T_VisuQVis.ptrT_ExchgParam^.T_SafetyCtrl.iMsgInfoLine3:=1;	(* WILL BE READY TO USE IT! *)
			T_VisuQVis.ptrT_ExchgParam^.T_SafetyCtrl.iMsgInfoLine4:=1;	(*  *)
			T_VisuQVis.ptrT_ExchgParam^.T_SafetyCtrl.xConfirmMsgInfo:=FALSE;
			T_VisuQVis.ptrT_ExchgParam^.T_SafetyCtrl.xBlockVisuObject:=TRUE;
			xRdy:=TRUE;
			(* next step *)
			iStepFunction:=985;
		985:	IF T_VisuQVis.ptrT_ExchgParam^.T_SafetyCtrl.xConfirmMsgInfo THEN
				T_VisuQVis.ptrT_ExchgParam^.T_SafetyCtrl.xBlockVisuObject:=FALSE;
				T_VisuQVis.ptrT_ExchgParam^.T_SafetyCtrl.bStateMessageInfo:=0;
				T_VisuQVis.ptrT_ExchgParam^.T_SafetyCtrl.xConfirmMsgInfo:=FALSE;
				T_VisuQVis.ptrT_ExchgParam^.T_SafetyCtrl.bStateAutoGeometry:=1;
				T_VisuQVis.ptrT_ExchgParam^.T_SafetyCtrl.bStateAutoGroove:=1;
				T_VisuQVis.ptrT_ExchgParam^.T_SafetyCtrl.bStateReference:=1;
				T_VisuQVis.ptrT_ExchgParam^.T_SafetyCtrl.bStateToolCalibration:=1;
				T_VisuQVis.ptrT_ExchgParam^.T_SafetyCtrl.bStateToolTorque:=1;
				T_VisuQVis.ptrT_ExchgParam^.T_SafetyCtrl.bStateTeachInToolLeft:=1;
				T_VisuQVis.ptrT_ExchgParam^.T_SafetyCtrl.bStateTeachInToolCenter:=1;
				T_VisuQVis.ptrT_ExchgParam^.T_SafetyCtrl.bStateTeachInToolRight:=1;
				T_VisuQVis.ptrT_ExchgParam^.T_SafetyCtrl.bStateTeachInToolFeeder:=1;
				T_VisuQVis.ptrT_ExchgParam^.T_SafetyCtrl.bStateTeachInGrindFeeder:=1;
				T_VisuQVis.ptrT_ExchgParam^.T_StationCommon.iWireFeederRefIndexState:=1;
				(* next step *)
				iStepFunction:=990;
			END_IF;
		(* End function *)
		990:	T_StartUp.T_State.xCompleted:=TRUE;
			T_StartUp.T_State.xBlockChangeMovementVisu:=FALSE;
			T_StartUp.T_State.xBlockVisuNavigation:=FALSE;
			T_VisuQVis.ptrT_ExchgParam^.T_SafetyCtrl.xBlockVisuObject:=FALSE;
			T_StartUp.T_Ctrle.xDone:=TRUE;
			T_StartUp.T_Ctrle.xErr:=FALSE;
			T_StartUp.T_Ctrle.udiErrorID:=16#0;
			xLoading:=FALSE;
			tTimeOutFunction:=T#0s;	(* deactivate the time out *)
		(* Error function, set output disable *)
		999:	tTimeOutFunction:=T#0s;	(* deactivate the time out *)
			T_Station.TControl.xEnable:=FALSE;
			T_VisuQVis.ptrT_ExchgParam^.T_Visu.iLoadingStartPage:=1;
			T_VisuQVis.ptrT_ExchgParam^.T_SafetyCtrl.iStateStartPage:=0;	(* No Text *)
			(* next step *)
			iStepFunction:=9994;
		9994:(* Overlay Message Error *)
			T_VisuQVis.ptrT_ExchgParam^.T_SafetyCtrl.bStateMessageError:=1;
			T_VisuQVis.ptrT_ExchgParam^.T_SafetyCtrl.bStateMessageInfo:=0;
			T_VisuQVis.ptrT_ExchgParam^.T_SafetyCtrl.bStateMessageWarning:=0;
			T_VisuQVis.ptrT_ExchgParam^.T_SafetyCtrl.iMsgErrorLine1:=7;	(* WHILE BOOTING THE MACHINE *)
			T_VisuQVis.ptrT_ExchgParam^.T_SafetyCtrl.iMsgErrorLine2:=7;	(* AN ERROR HAS OCCURRED *)
			T_VisuQVis.ptrT_ExchgParam^.T_SafetyCtrl.iMsgErrorLine3:=7;	(* PLEASE CONFIRM AND CHECK *)
			T_VisuQVis.ptrT_ExchgParam^.T_SafetyCtrl.iMsgErrorLine4:=7;	(* THE ACCORDING ERROR *)
			T_VisuQVis.ptrT_ExchgParam^.T_SafetyCtrl.xConfirmMsgError:=FALSE;
			T_VisuQVis.ptrT_ExchgParam^.T_SafetyCtrl.xBlockVisuObject:=TRUE;
			T_TwinSafeCtrleOUT.xTwinSAFE_Run:=FALSE;	(* Stop TwinSafe Groupe *)
			(* next step *)
			iStepFunction:=9995;
		9995:IF T_VisuQVis.ptrT_ExchgParam^.T_SafetyCtrl.xConfirmMsgError THEN
				T_VisuQVis.ptrT_ExchgParam^.T_SafetyCtrl.xBlockVisuObject:=FALSE;
				T_VisuQVis.ptrT_ExchgParam^.T_SafetyCtrl.bStateMessageError:=0;
				T_VisuQVis.ptrT_ExchgParam^.T_SafetyCtrl.xConfirmMsgError:=FALSE;
				(* next step *)
				iStepFunction:=9996;
			END_IF;
		9996:	xLoading:=FALSE;
				xStartBooting:=TRUE;
				tTimeOutFunction:=T#0s;	(* deactivate the time out *)
				(* next step *)
				iStepFunction:=1;
		END_CASE
	END_IF;
(****************************************************************************************************************************************************)
(***********                                                      start of the execution for the function of the start up                                                          ************)
(****************************************************************************************************************************************************)

(* Control Lamp for the power supply of the Ecostep *)
	IF NOT(T_TwinSafeIn.IxPowerSupplyEcoStep) THEN
		QarxDigitalOutput[4]:=TRUE;	(* QxCtrlLampCurEcoButton *)
		T_VisuQVis.ptrT_ExchgParam^.T_SafetyCtrl.iStateStartPage:=4;	(* Message: Release AxesCurrentButton *)
	ELSE
		QarxDigitalOutput[4]:=FALSE;	(* QxCtrlLampCurEcoButton *)
	END_IF;

